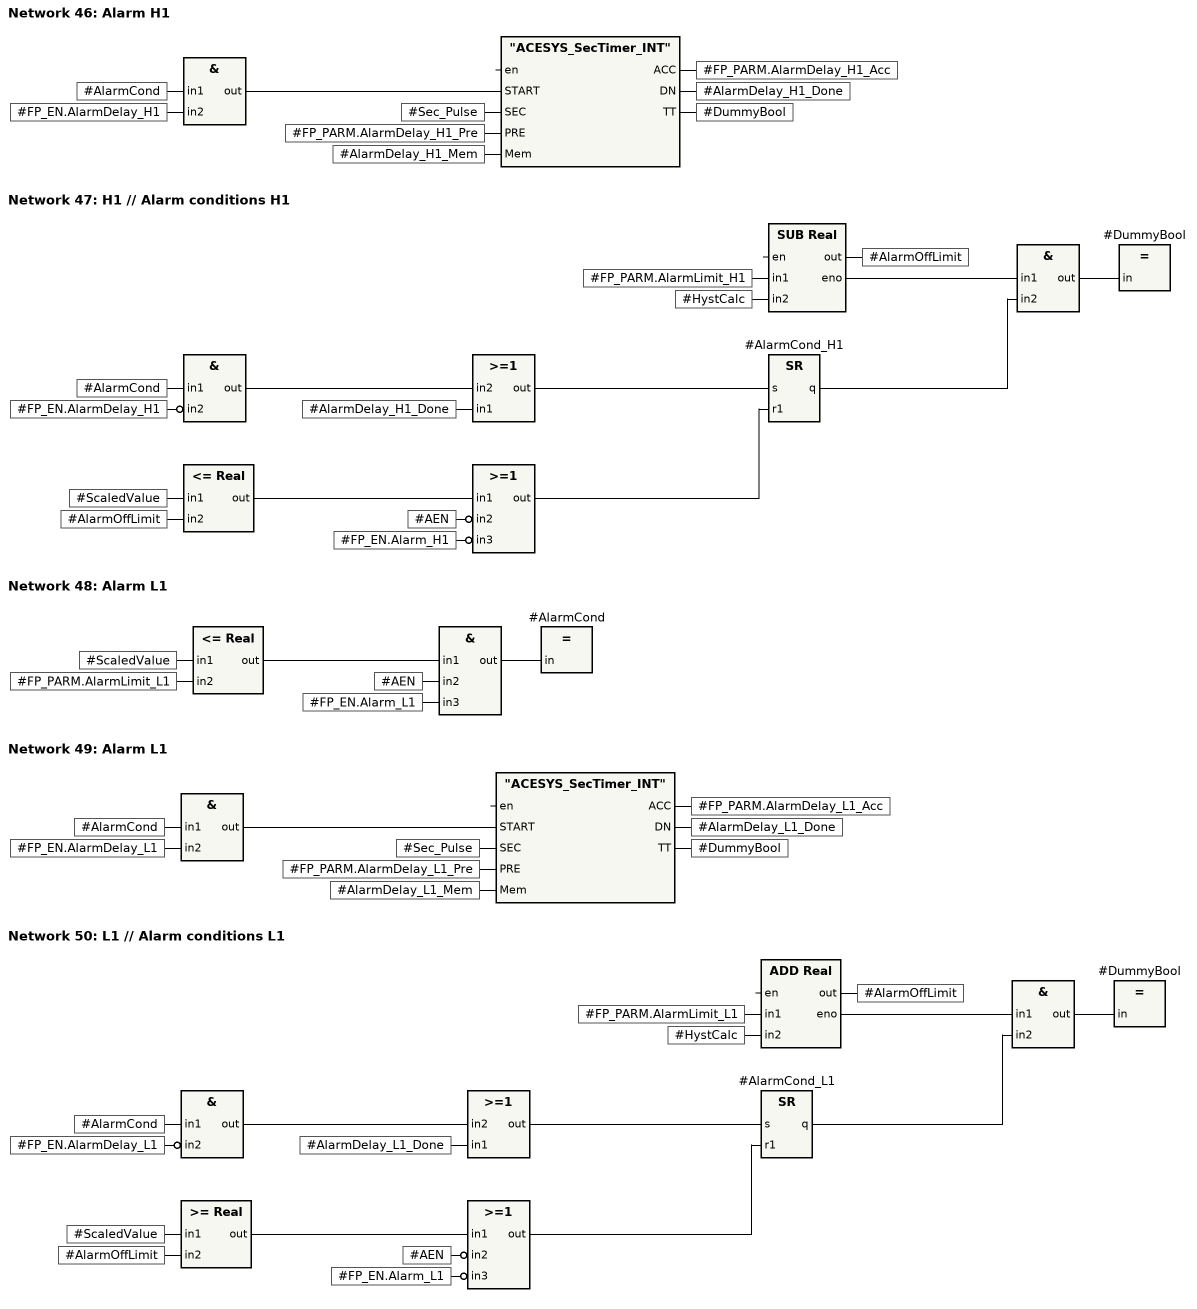
   "ACESYS_SecTimer_INT"(START := #AlarmCond AND #FP_EN.AlarmDelay_H1,
                         SEC := #Sec_Pulse,
                         PRE := #FP_PARM.AlarmDelay_H1_Pre,
                         Mem := #AlarmDelay_H1_Mem,
                         ACC => #FP_PARM.AlarmDelay_H1_Acc,
                         DN => #AlarmDelay_H1_Done,
                         TT => #DummyBool);
END_REGION

REGION Network 47: H1 // Alarm conditions H1
   // ENO of a box is taken as its EN; it also drops when the box reports an error
   #AlarmOffLimit := #FP_PARM.AlarmLimit_H1 - #HystCalc;
   IF (#AlarmCond AND NOT #FP_EN.AlarmDelay_H1) OR #AlarmDelay_H1_Done THEN
       #AlarmCond_H1 := TRUE;   // SR flip-flop
   END_IF;
   IF (#ScaledValue <= #AlarmOffLimit) OR NOT #AEN OR NOT #FP_EN.Alarm_H1 THEN
       #AlarmCond_H1 := FALSE;
   END_IF;
   #DummyBool := #AlarmCond_H1;
END_REGION

REGION Network 48: Alarm L1
   #AlarmCond := (#ScaledValue <= #FP_PARM.AlarmLimit_L1) AND #AEN AND #FP_EN.Alarm_L1;
END_REGION

REGION Network 49: Alarm L1
   "ACESYS_SecTimer_INT"(START := #AlarmCond AND #FP_EN.AlarmDelay_L1,
                         SEC := #Sec_Pulse,
                         PRE := #FP_PARM.AlarmDelay_L1_Pre,
                         Mem := #AlarmDelay_L1_Mem,
                         ACC => #FP_PARM.AlarmDelay_L1_Acc,
                         DN => #AlarmDelay_L1_Done,
                         TT => #DummyBool);
END_REGION

REGION Network 50: L1 // Alarm conditions L1
   // ENO of a box is taken as its EN; it also drops when the box reports an error
   #AlarmOffLimit := #FP_PARM.AlarmLimit_L1 + #HystCalc;
   IF (#AlarmCond AND NOT #FP_EN.AlarmDelay_L1) OR #AlarmDelay_L1_Done THEN
       #AlarmCond_L1 := TRUE;   // SR flip-flop
   END_IF;
   IF (#ScaledValue >= #AlarmOffLimit) OR NOT #AEN OR NOT #FP_EN.Alarm_L1 THEN
       #AlarmCond_L1 := FALSE;
   END_IF;
   #DummyBool := #AlarmCond_L1;
END_REGION

REGION Network 51: Alarm L2
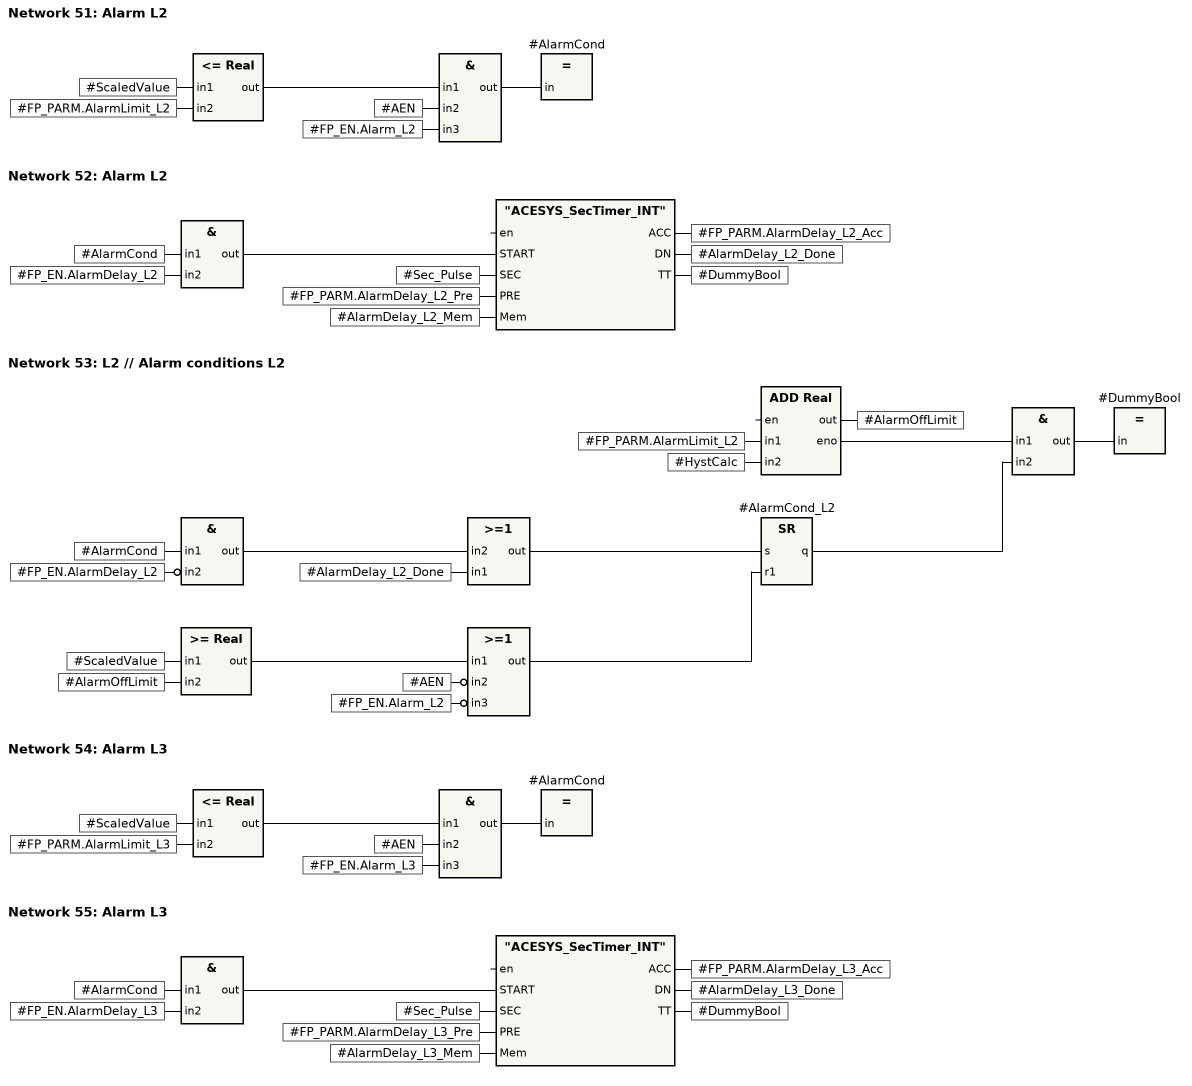
   #AlarmCond := (#ScaledValue <= #FP_PARM.AlarmLimit_L2) AND #AEN AND #FP_EN.Alarm_L2;
END_REGION

REGION Network 52: Alarm L2
   "ACESYS_SecTimer_INT"(START := #AlarmCond AND #FP_EN.AlarmDelay_L2,
                         SEC := #Sec_Pulse,
                         PRE := #FP_PARM.AlarmDelay_L2_Pre,
                         Mem := #AlarmDelay_L2_Mem,
                         ACC => #FP_PARM.AlarmDelay_L2_Acc,
                         DN => #AlarmDelay_L2_Done,
                         TT => #DummyBool);
END_REGION

REGION Network 53: L2 // Alarm conditions L2
   // ENO of a box is taken as its EN; it also drops when the box reports an error
   #AlarmOffLimit := #FP_PARM.AlarmLimit_L2 + #HystCalc;
   IF (#AlarmCond AND NOT #FP_EN.AlarmDelay_L2) OR #AlarmDelay_L2_Done THEN
       #AlarmCond_L2 := TRUE;   // SR flip-flop
   END_IF;
   IF (#ScaledValue >= #AlarmOffLimit) OR NOT #AEN OR NOT #FP_EN.Alarm_L2 THEN
       #AlarmCond_L2 := FALSE;
   END_IF;
   #DummyBool := #AlarmCond_L2;
END_REGION

REGION Network 54: Alarm L3
   #AlarmCond := (#ScaledValue <= #FP_PARM.AlarmLimit_L3) AND #AEN AND #FP_EN.Alarm_L3;
END_REGION

REGION Network 55: Alarm L3
   "ACESYS_SecTimer_INT"(START := #AlarmCond AND #FP_EN.AlarmDelay_L3,
                         SEC := #Sec_Pulse,
                         PRE := #FP_PARM.AlarmDelay_L3_Pre,
                         Mem := #AlarmDelay_L3_Mem,
                         ACC => #FP_PARM.AlarmDelay_L3_Acc,
                         DN => #AlarmDelay_L3_Done,
                         TT => #DummyBool);
END_REGION

REGION Network 56: L3 // Alarm conditions L3
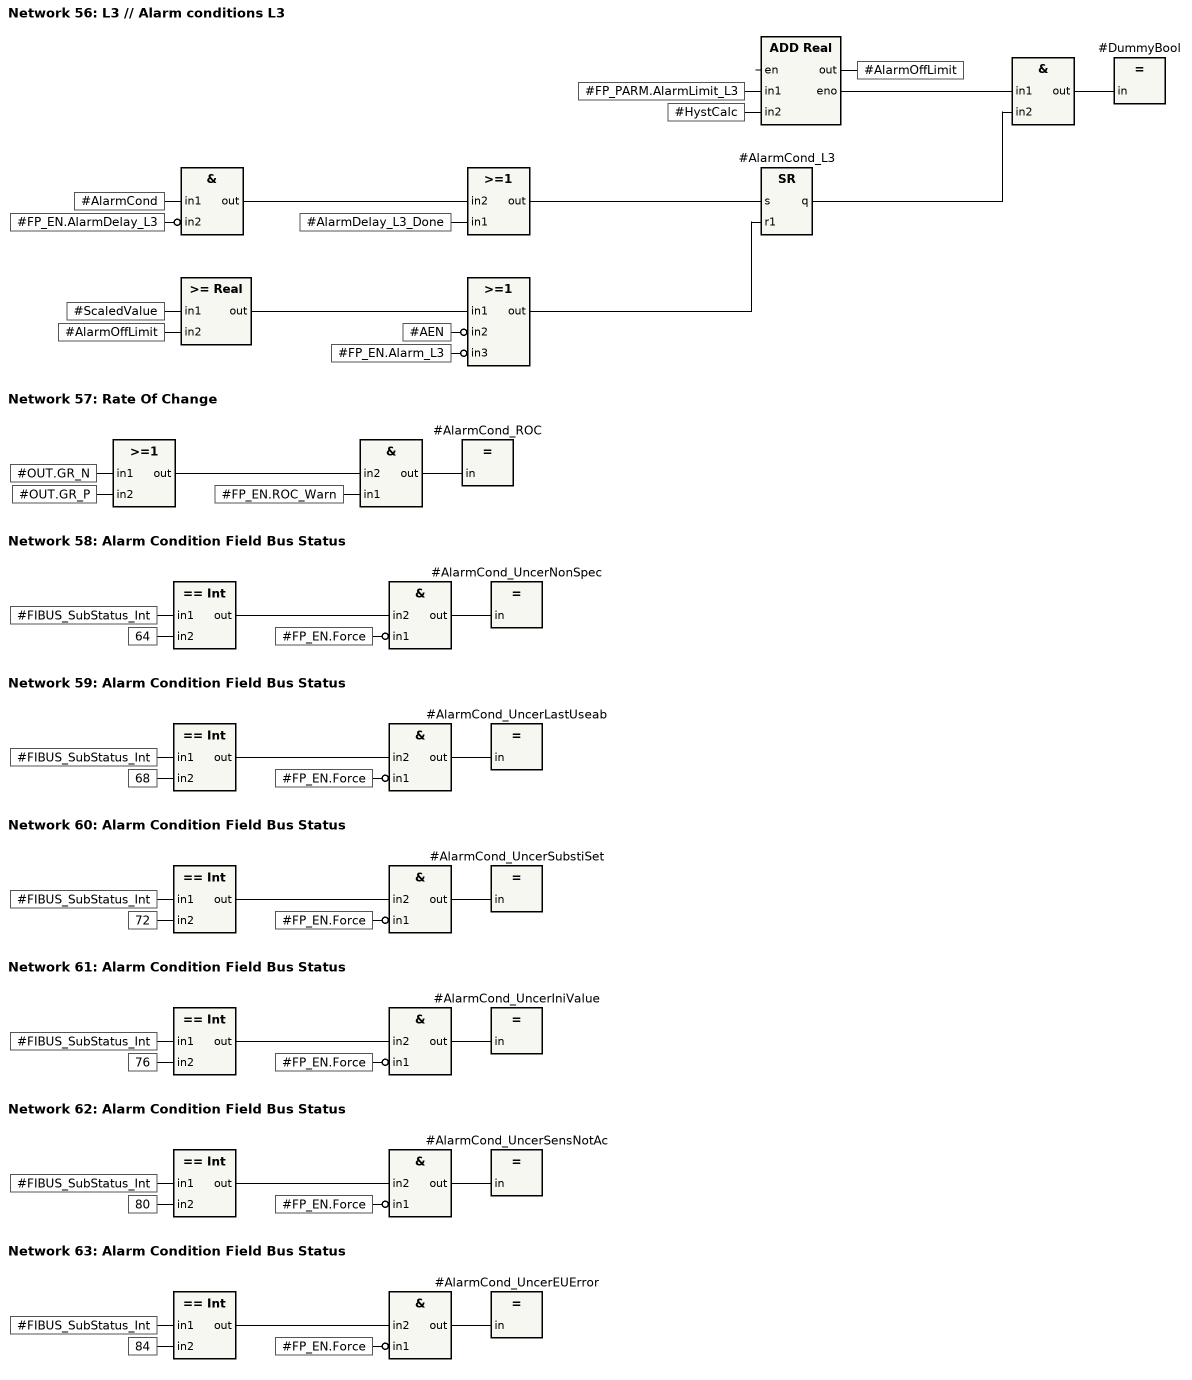
   // ENO of a box is taken as its EN; it also drops when the box reports an error
   #AlarmOffLimit := #FP_PARM.AlarmLimit_L3 + #HystCalc;
   IF (#AlarmCond AND NOT #FP_EN.AlarmDelay_L3) OR #AlarmDelay_L3_Done THEN
       #AlarmCond_L3 := TRUE;   // SR flip-flop
   END_IF;
   IF (#ScaledValue >= #AlarmOffLimit) OR NOT #AEN OR NOT #FP_EN.Alarm_L3 THEN
       #AlarmCond_L3 := FALSE;
   END_IF;
   #DummyBool := #AlarmCond_L3;
END_REGION

REGION Network 57: Rate Of Change
   // >>>>>Rate Of Change (RAC)<<<<<
   // 
   // Warning only
   #AlarmCond_ROC := (#OUT.GR_N OR #OUT.GR_P) AND #FP_EN.ROC_Warn;
END_REGION

REGION Network 58: Alarm Condition Field Bus Status
   // Build 003 - 24 Oct 2019 : FP_En_Force flag added
   #AlarmCond_UncerNonSpec := (#FIBUS_SubStatus_Int = 64) AND NOT #FP_EN.Force;
END_REGION

REGION Network 59: Alarm Condition Field Bus Status
   // Build 003 - 24 Oct 2019 : FP_En_Force flag added
   #AlarmCond_UncerLastUseab := (#FIBUS_SubStatus_Int = 68) AND NOT #FP_EN.Force;
END_REGION

REGION Network 60: Alarm Condition Field Bus Status
   // Build 003 - 24 Oct 2019 : FP_En_Force flag added
   #AlarmCond_UncerSubstiSet := (#FIBUS_SubStatus_Int = 72) AND NOT #FP_EN.Force;
END_REGION

REGION Network 61: Alarm Condition Field Bus Status
   // Build 003 - 24 Oct 2019 : FP_En_Force flag added
   #AlarmCond_UncerIniValue := (#FIBUS_SubStatus_Int = 76) AND NOT #FP_EN.Force;
END_REGION

REGION Network 62: Alarm Condition Field Bus Status
   // Build 003 - 24 Oct 2019 : FP_En_Force flag added
   #AlarmCond_UncerSensNotAc := (#FIBUS_SubStatus_Int = 80) AND NOT #FP_EN.Force;
END_REGION

REGION Network 63: Alarm Condition Field Bus Status
   #AlarmCond_UncerEUError := (#FIBUS_SubStatus_Int = 84) AND NOT #FP_EN.Force;
END_REGION

REGION Network 64: Alarm Condition Field Bus Status
   // Build 003 - 24 Oct 2019 : FP_En_Force flag added
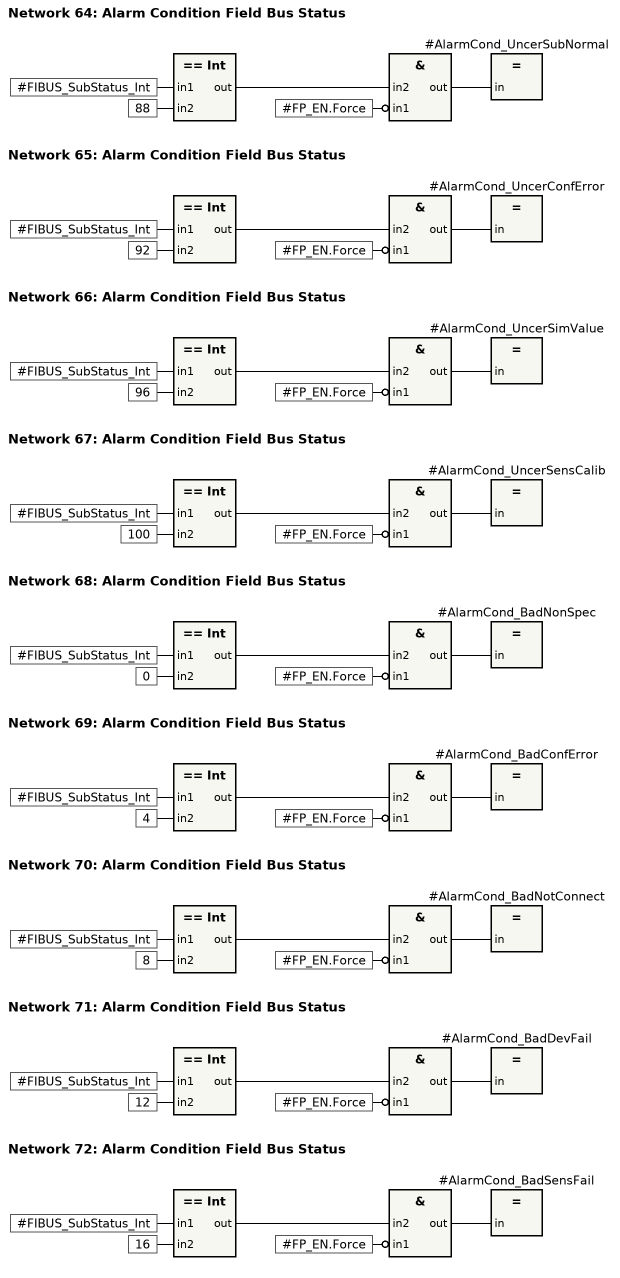
   #AlarmCond_UncerSubNormal := (#FIBUS_SubStatus_Int = 88) AND NOT #FP_EN.Force;
END_REGION

REGION Network 65: Alarm Condition Field Bus Status
   #AlarmCond_UncerConfError := (#FIBUS_SubStatus_Int = 92) AND NOT #FP_EN.Force;
END_REGION

REGION Network 66: Alarm Condition Field Bus Status
   #AlarmCond_UncerSimValue := (#FIBUS_SubStatus_Int = 96) AND NOT #FP_EN.Force;
END_REGION

REGION Network 67: Alarm Condition Field Bus Status
   // Build 003 - 24 Oct 2019 : FP_En_Force flag added
   #AlarmCond_UncerSensCalib := (#FIBUS_SubStatus_Int = 100) AND NOT #FP_EN.Force;
END_REGION

REGION Network 68: Alarm Condition Field Bus Status
   #AlarmCond_BadNonSpec := (#FIBUS_SubStatus_Int = 0) AND NOT #FP_EN.Force;
END_REGION

REGION Network 69: Alarm Condition Field Bus Status
   // Build 003 - 24 Oct 2019 : FP_En_Force flag added
   #AlarmCond_BadConfError := (#FIBUS_SubStatus_Int = 4) AND NOT #FP_EN.Force;
END_REGION

REGION Network 70: Alarm Condition Field Bus Status
   #AlarmCond_BadNotConnect := (#FIBUS_SubStatus_Int = 8) AND NOT #FP_EN.Force;
END_REGION

REGION Network 71: Alarm Condition Field Bus Status
   // Build 003 - 24 Oct 2019 : FP_En_Force flag added
   #AlarmCond_BadDevFail := (#FIBUS_SubStatus_Int = 12) AND NOT #FP_EN.Force;
END_REGION

REGION Network 72: Alarm Condition Field Bus Status
   // Build 003 - 24 Oct 2019 : FP_En_Force flag added
   #AlarmCond_BadSensFail := (#FIBUS_SubStatus_Int = 16) AND NOT #FP_EN.Force;
END_REGION

REGION Network 73: Alarm Condition Field Bus Status
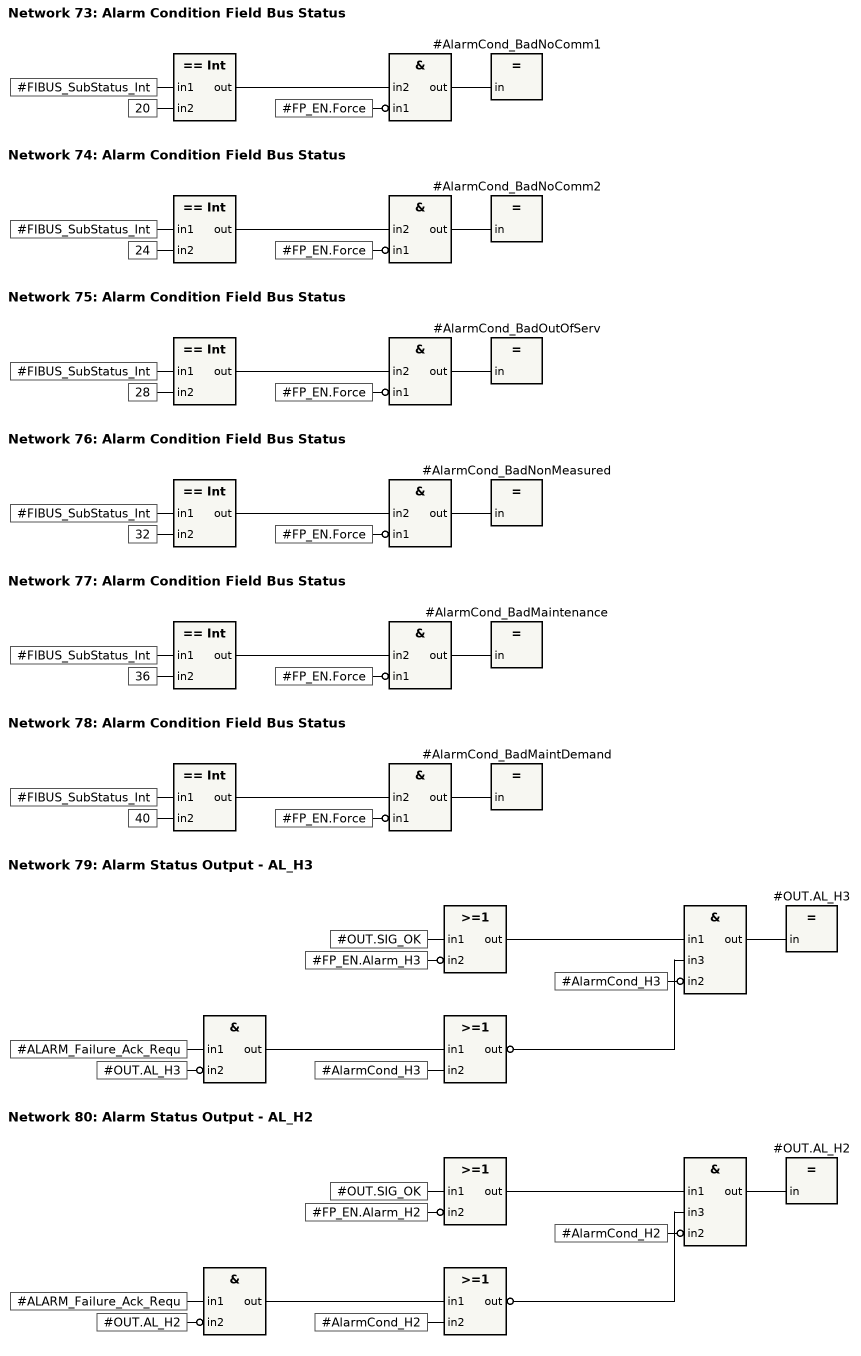
   #AlarmCond_BadNoComm1 := (#FIBUS_SubStatus_Int = 20) AND NOT #FP_EN.Force;
END_REGION

REGION Network 74: Alarm Condition Field Bus Status
   // Build 003 - 24 Oct 2019 : FP_En_Force flag added
   #AlarmCond_BadNoComm2 := (#FIBUS_SubStatus_Int = 24) AND NOT #FP_EN.Force;
END_REGION

REGION Network 75: Alarm Condition Field Bus Status
   #AlarmCond_BadOutOfServ := (#FIBUS_SubStatus_Int = 28) AND NOT #FP_EN.Force;
END_REGION

REGION Network 76: Alarm Condition Field Bus Status
   // Build 003 - 24 Oct 2019 : FP_En_Force flag added
   #AlarmCond_BadNonMeasured := (#FIBUS_SubStatus_Int = 32) AND NOT #FP_EN.Force;
END_REGION

REGION Network 77: Alarm Condition Field Bus Status
   // Build 003 - 24 Oct 2019 : FP_En_Force flag added
   #AlarmCond_BadMaintenance := (#FIBUS_SubStatus_Int = 36) AND NOT #FP_EN.Force;
END_REGION

REGION Network 78: Alarm Condition Field Bus Status
   // Build 003 - 24 Oct 2019 : FP_En_Force flag added
   #AlarmCond_BadMaintDemand := (#FIBUS_SubStatus_Int = 40) AND NOT #FP_EN.Force;
END_REGION

REGION Network 79: Alarm Status Output - AL_H3
   #OUT.AL_H3 := (#OUT.SIG_OK OR NOT #FP_EN.Alarm_H3) AND NOT ((#ALARM_Failure_Ack_Requ AND NOT #OUT.AL_H3) OR #AlarmCond_H3) AND NOT #AlarmCond_H3;
END_REGION

REGION Network 80: Alarm Status Output - AL_H2
   #OUT.AL_H2 := (#OUT.SIG_OK OR NOT #FP_EN.Alarm_H2) AND NOT ((#ALARM_Failure_Ack_Requ AND NOT #OUT.AL_H2) OR #AlarmCond_H2) AND NOT #AlarmCond_H2;
END_REGION

REGION Network 81: Alarm Status Output - AL_H1
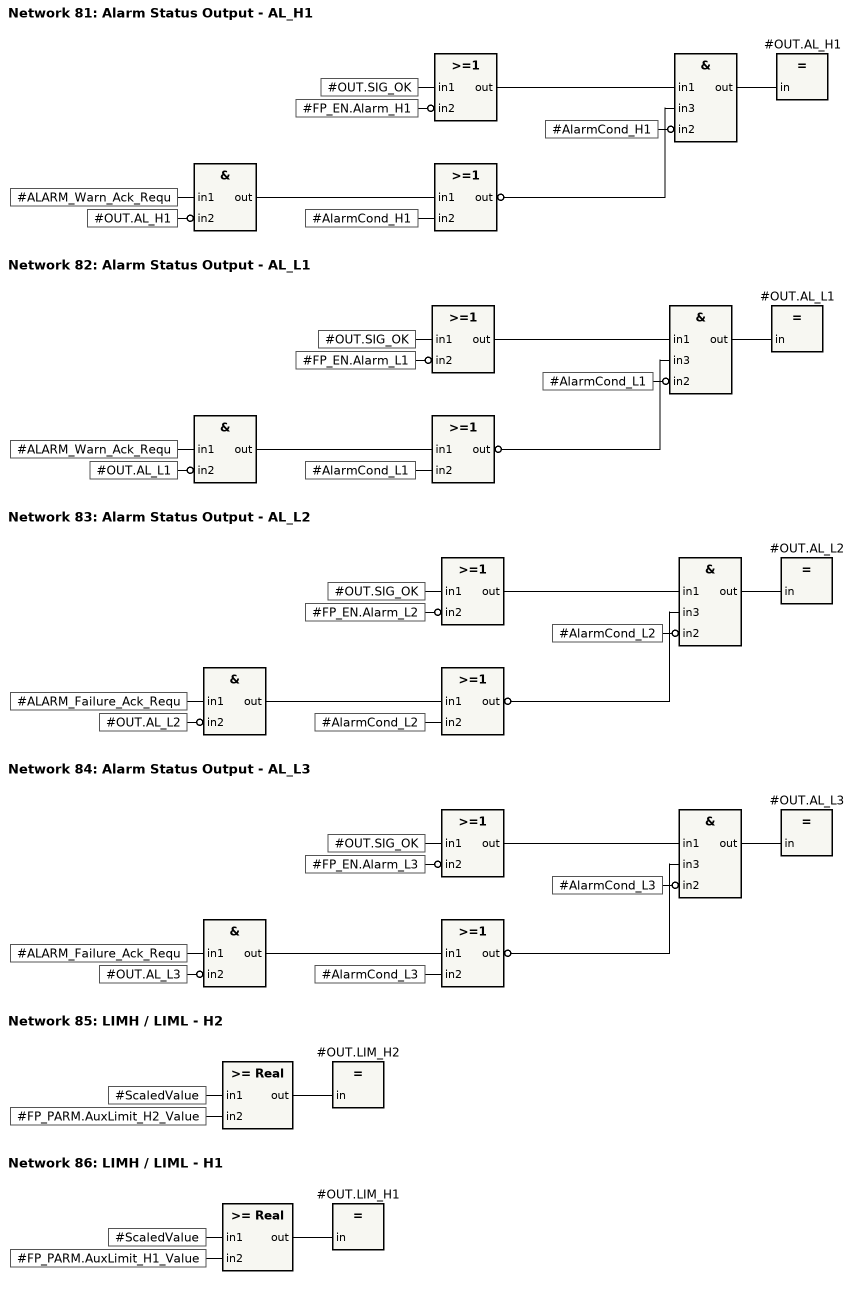
   #OUT.AL_H1 := (#OUT.SIG_OK OR NOT #FP_EN.Alarm_H1) AND NOT ((#ALARM_Warn_Ack_Requ AND NOT #OUT.AL_H1) OR #AlarmCond_H1) AND NOT #AlarmCond_H1;
END_REGION

REGION Network 82: Alarm Status Output - AL_L1
   #OUT.AL_L1 := (#OUT.SIG_OK OR NOT #FP_EN.Alarm_L1) AND NOT ((#ALARM_Warn_Ack_Requ AND NOT #OUT.AL_L1) OR #AlarmCond_L1) AND NOT #AlarmCond_L1;
END_REGION

REGION Network 83: Alarm Status Output - AL_L2
   #OUT.AL_L2 := (#OUT.SIG_OK OR NOT #FP_EN.Alarm_L2) AND NOT ((#ALARM_Failure_Ack_Requ AND NOT #OUT.AL_L2) OR #AlarmCond_L2) AND NOT #AlarmCond_L2;
END_REGION

REGION Network 84: Alarm Status Output - AL_L3
   #OUT.AL_L3 := (#OUT.SIG_OK OR NOT #FP_EN.Alarm_L3) AND NOT ((#ALARM_Failure_Ack_Requ AND NOT #OUT.AL_L3) OR #AlarmCond_L3) AND NOT #AlarmCond_L3;
END_REGION

REGION Network 85: LIMH / LIML - H2
   #OUT.LIM_H2 := #ScaledValue >= #FP_PARM.AuxLimit_H2_Value;
END_REGION

REGION Network 86: LIMH / LIML - H1
   #OUT.LIM_H1 := #ScaledValue >= #FP_PARM.AuxLimit_H1_Value;
END_REGION

REGION Network 87: LIMH / LIML - L1
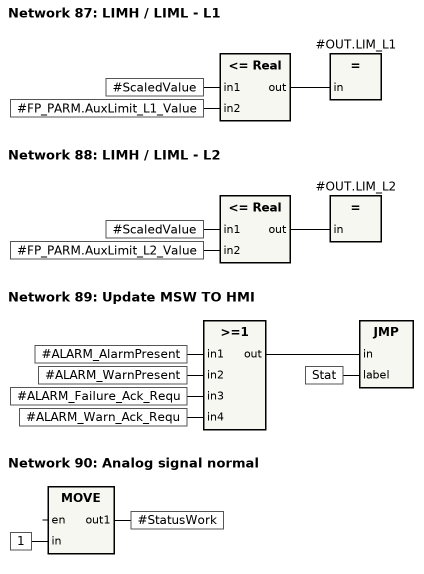
   #OUT.LIM_L1 := #ScaledValue <= #FP_PARM.AuxLimit_L1_Value;
END_REGION

REGION Network 88: LIMH / LIML - L2
   #OUT.LIM_L2 := #ScaledValue <= #FP_PARM.AuxLimit_L2_Value;
END_REGION

REGION Network 89: Update MSW TO HMI
   // Stat = Skip Sensor Status
   IF #ALARM_AlarmPresent OR #ALARM_WarnPresent OR #ALARM_Failure_Ack_Requ OR #ALARM_Warn_Ack_Requ THEN
       GOTO Stat;
   END_IF;
END_REGION

REGION Network 90: Analog signal normal
   #StatusWork := 1;
END_REGION

REGION Network 91: Report Good status
   // 132 = Active block alarm
   // 136 = Active advisory alarm
   // 140 = Active critical alarm
   // 144 = Unacknowledged block alarm
   // 148 = Unacknowledged advisory alarm
   // 152 = Unacknowledged critical alarm
   // 156 = Not used
   // 160 = Init fail safe
   // 164 = Maintenance required
   // 
   // Build 006 - 22 Nov 2017 : Status work changed from 132 - 164 to 50 - 57
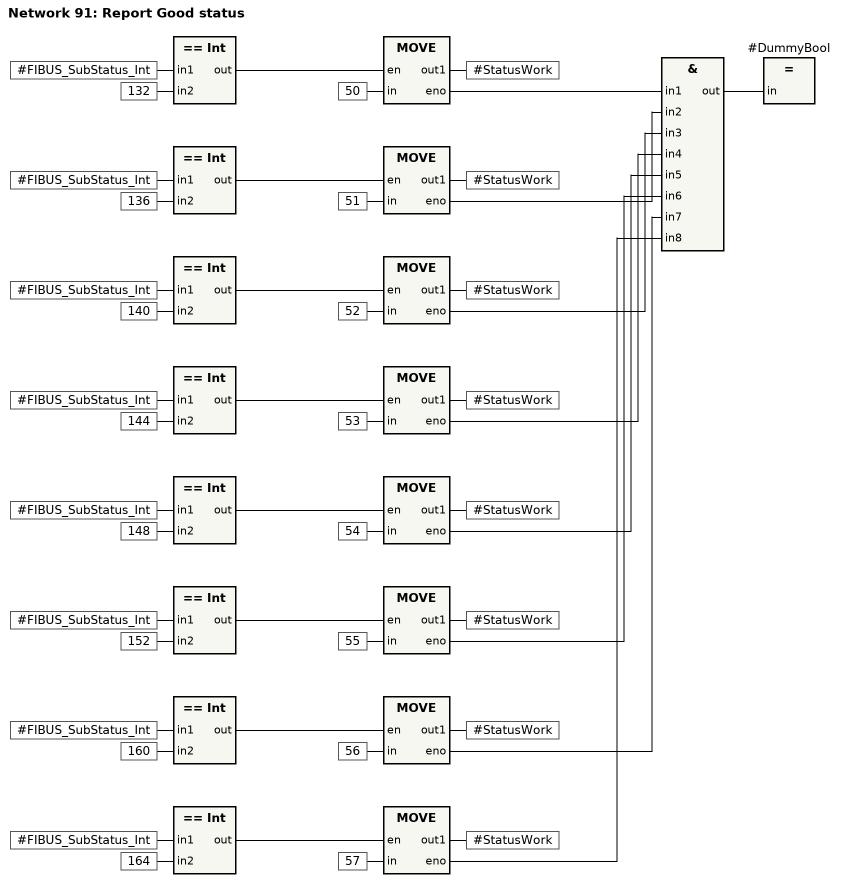
   // ENO of a box is taken as its EN; it also drops when the box reports an error
   #_w1 := #FIBUS_SubStatus_Int = 132;
   IF #_w1 THEN #StatusWork := 50; END_IF;
   #_w2 := #FIBUS_SubStatus_Int = 136;
   IF #_w2 THEN #StatusWork := 51; END_IF;
   #_w3 := #FIBUS_SubStatus_Int = 140;
   IF #_w3 THEN #StatusWork := 52; END_IF;
   #_w4 := #FIBUS_SubStatus_Int = 144;
   IF #_w4 THEN #StatusWork := 53; END_IF;
   #_w5 := #FIBUS_SubStatus_Int = 148;
   IF #_w5 THEN #StatusWork := 54; END_IF;
   #_w6 := #FIBUS_SubStatus_Int = 152;
   IF #_w6 THEN #StatusWork := 55; END_IF;
   #_w7 := #FIBUS_SubStatus_Int = 160;
   IF #_w7 THEN #StatusWork := 56; END_IF;
   #_w8 := #FIBUS_SubStatus_Int = 164;
   IF #_w8 THEN #StatusWork := 57; END_IF;
   #DummyBool := #_w1 AND #_w2 AND #_w3 AND #_w4 AND #_w5 AND #_w6 AND #_w7 AND #_w8;
END_REGION

REGION Network 92: Jump Network
   // >>>>>SIGNAL VALID DETECTION<<<<<
   // 
   // Jump destination if ignore sensor Status
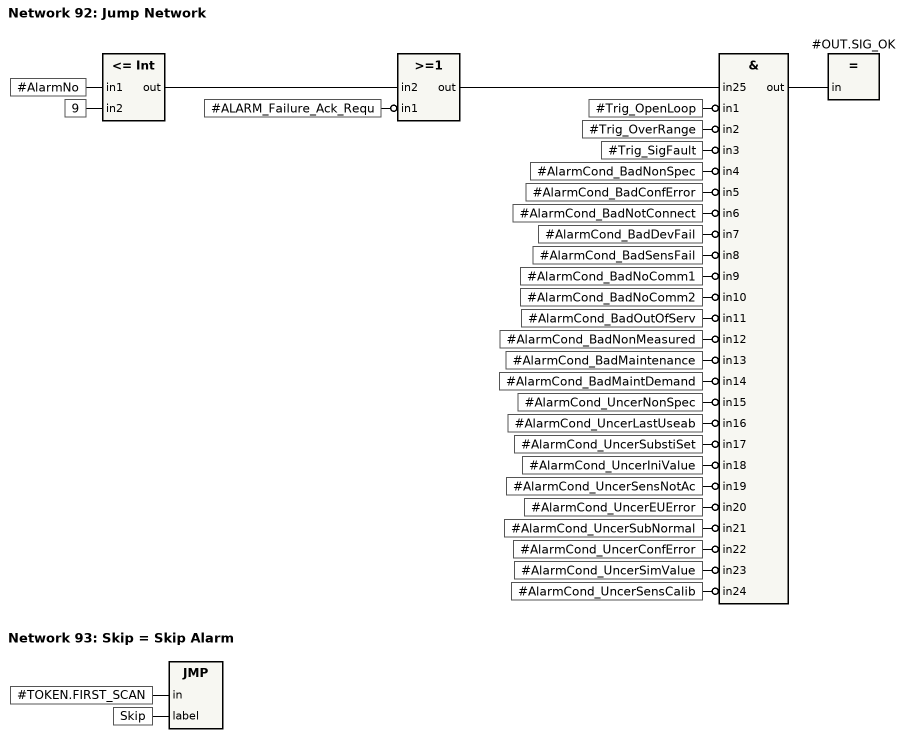
   Stat:
   #OUT.SIG_OK := ((#AlarmNo <= 9) OR NOT #ALARM_Failure_Ack_Requ) AND NOT #Trig_OpenLoop AND NOT #Trig_OverRange AND NOT #Trig_SigFault AND NOT #AlarmCond_BadNonSpec AND NOT #AlarmCond_BadConfError AND NOT #AlarmCond_BadNotConnect AND NOT #AlarmCond_BadDevFail AND NOT #AlarmCond_BadSensFail AND NOT #AlarmCond_BadNoComm1 AND NOT #AlarmCond_BadNoComm2 AND NOT #AlarmCond_BadOutOfServ AND NOT #AlarmCond_BadNonMeasured AND NOT #AlarmCond_BadMaintenance AND NOT #AlarmCond_BadMaintDemand AND NOT #AlarmCond_UncerNonSpec AND NOT #AlarmCond_UncerLastUseab AND NOT #AlarmCond_UncerSubstiSet AND NOT #AlarmCond_UncerIniValue AND NOT #AlarmCond_UncerSensNotAc AND NOT #AlarmCond_UncerEUError AND NOT #AlarmCond_UncerSubNormal AND NOT #AlarmCond_UncerConfError AND NOT #AlarmCond_UncerSimValue AND NOT #AlarmCond_UncerSensCalib;
END_REGION

REGION Network 93: Skip = Skip Alarm
   // >>>>>Alarm Present<<<<<
   // 
   // Skip = Skip Alarm
   IF #TOKEN.FIRST_SCAN THEN GOTO Skip; END_IF;
END_REGION

REGION Network 94: Alarm
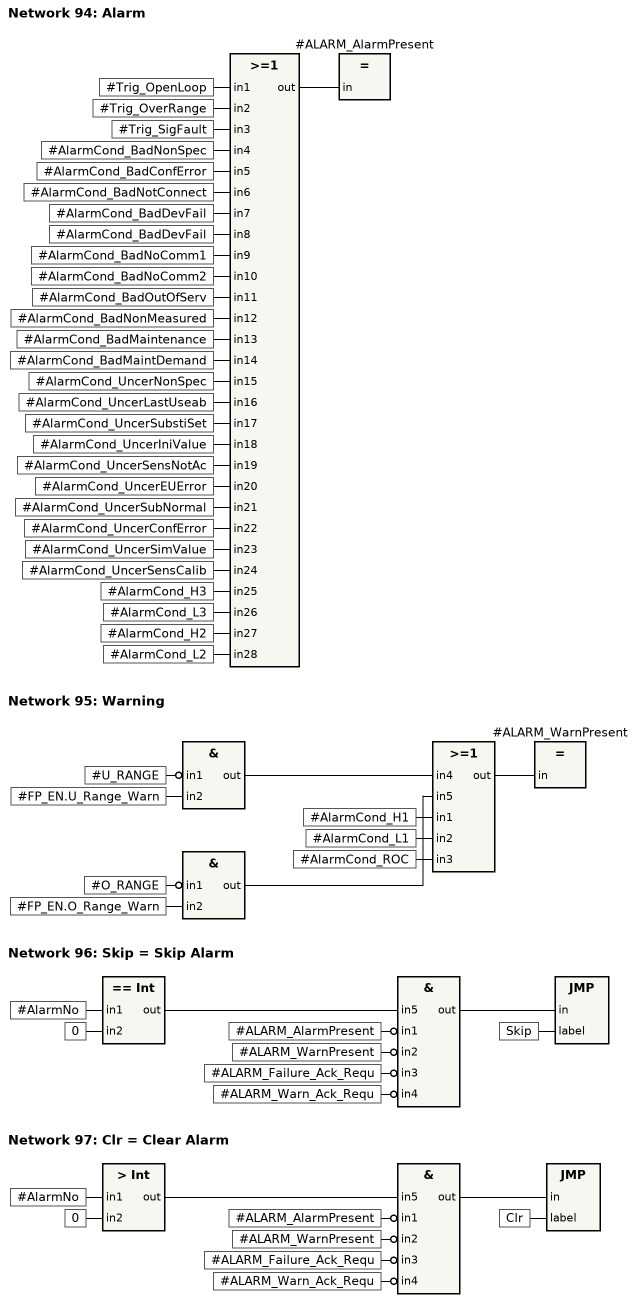
   #ALARM_AlarmPresent := #Trig_OpenLoop OR #Trig_OverRange OR #Trig_SigFault OR #AlarmCond_BadNonSpec OR #AlarmCond_BadConfError OR #AlarmCond_BadNotConnect OR #AlarmCond_BadDevFail OR #AlarmCond_BadDevFail OR #AlarmCond_BadNoComm1 OR #AlarmCond_BadNoComm2 OR #AlarmCond_BadOutOfServ OR #AlarmCond_BadNonMeasured OR #AlarmCond_BadMaintenance OR #AlarmCond_BadMaintDemand OR #AlarmCond_UncerNonSpec OR #AlarmCond_UncerLastUseab OR #AlarmCond_UncerSubstiSet OR #AlarmCond_UncerIniValue OR #AlarmCond_UncerSensNotAc OR #AlarmCond_UncerEUError OR #AlarmCond_UncerSubNormal OR #AlarmCond_UncerConfError OR #AlarmCond_UncerSimValue OR #AlarmCond_UncerSensCalib OR #AlarmCond_H3 OR #AlarmCond_L3 OR #AlarmCond_H2 OR #AlarmCond_L2;
END_REGION

REGION Network 95: Warning
   #ALARM_WarnPresent := (NOT #U_RANGE AND #FP_EN.U_Range_Warn) OR (NOT #O_RANGE AND #FP_EN.O_Range_Warn) OR #AlarmCond_H1 OR #AlarmCond_L1 OR #AlarmCond_ROC;
END_REGION

REGION Network 96: Skip = Skip Alarm
   IF (#AlarmNo = 0) AND NOT #ALARM_AlarmPresent AND NOT #ALARM_WarnPresent AND NOT #ALARM_Failure_Ack_Requ AND NOT #ALARM_Warn_Ack_Requ THEN
       GOTO Skip;
   END_IF;
END_REGION

REGION Network 97: Clr = Clear Alarm
   IF (#AlarmNo > 0) AND NOT #ALARM_AlarmPresent AND NOT #ALARM_WarnPresent AND NOT #ALARM_Failure_Ack_Requ AND NOT #ALARM_Warn_Ack_Requ THEN
       GOTO Clr;
   END_IF;
END_REGION

REGION Network 98: Ack = Alarm Acknowledge
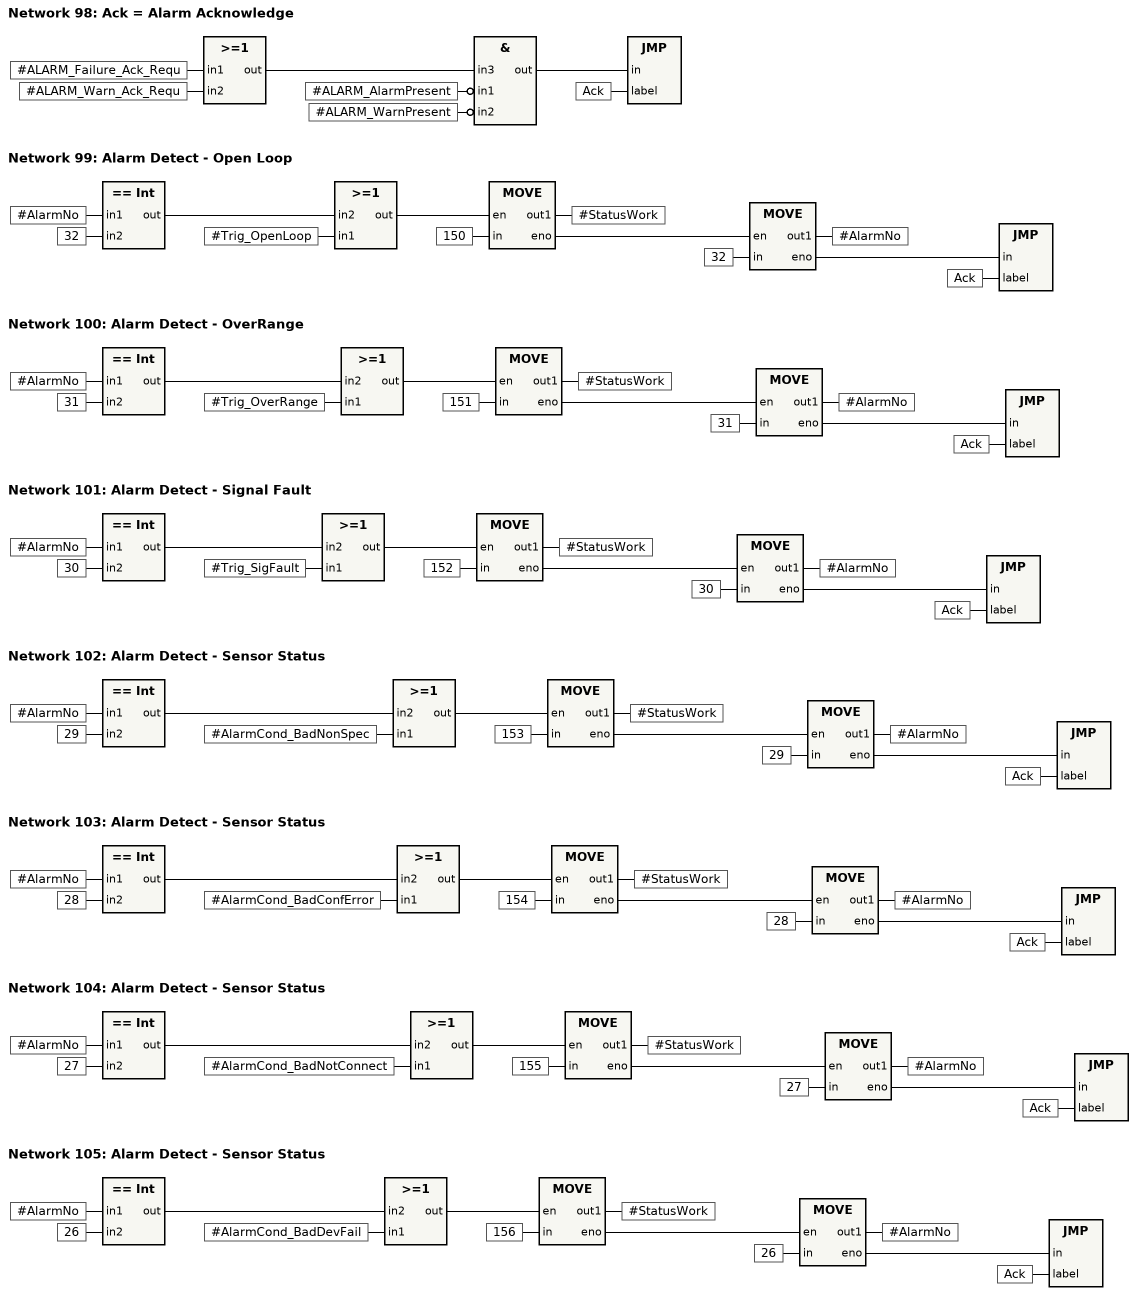
   IF (#ALARM_Failure_Ack_Requ OR #ALARM_Warn_Ack_Requ) AND NOT #ALARM_AlarmPresent AND NOT #ALARM_WarnPresent THEN
       GOTO Ack;
   END_IF;
END_REGION

REGION Network 99: Alarm Detect - Open Loop
   // ENO of a box is taken as its EN; it also drops when the box reports an error
   #_w1 := (#AlarmNo = 32) OR #Trig_OpenLoop;
   IF #_w1 THEN
       #StatusWork := 150;
       #AlarmNo := 32;
       GOTO Ack;
   END_IF;
END_REGION

REGION Network 100: Alarm Detect - OverRange
   // ENO of a box is taken as its EN; it also drops when the box reports an error
   #_w1 := (#AlarmNo = 31) OR #Trig_OverRange;
   IF #_w1 THEN
       #StatusWork := 151;
       #AlarmNo := 31;
       GOTO Ack;
   END_IF;
END_REGION

REGION Network 101: Alarm Detect - Signal Fault
   // ENO of a box is taken as its EN; it also drops when the box reports an error
   #_w1 := (#AlarmNo = 30) OR #Trig_SigFault;
   IF #_w1 THEN
       #StatusWork := 152;
       #AlarmNo := 30;
       GOTO Ack;
   END_IF;
END_REGION

REGION Network 102: Alarm Detect - Sensor Status
   // ENO of a box is taken as its EN; it also drops when the box reports an error
   #_w1 := (#AlarmNo = 29) OR #AlarmCond_BadNonSpec;
   IF #_w1 THEN
       #StatusWork := 153;
       #AlarmNo := 29;
       GOTO Ack;
   END_IF;
END_REGION

REGION Network 103: Alarm Detect - Sensor Status
   // ENO of a box is taken as its EN; it also drops when the box reports an error
   #_w1 := (#AlarmNo = 28) OR #AlarmCond_BadConfError;
   IF #_w1 THEN
       #StatusWork := 154;
       #AlarmNo := 28;
       GOTO Ack;
   END_IF;
END_REGION

REGION Network 104: Alarm Detect - Sensor Status
   // ENO of a box is taken as its EN; it also drops when the box reports an error
   #_w1 := (#AlarmNo = 27) OR #AlarmCond_BadNotConnect;
   IF #_w1 THEN
       #StatusWork := 155;
       #AlarmNo := 27;
       GOTO Ack;
   END_IF;
END_REGION

REGION Network 105: Alarm Detect - Sensor Status
   // ENO of a box is taken as its EN; it also drops when the box reports an error
   #_w1 := (#AlarmNo = 26) OR #AlarmCond_BadDevFail;
   IF #_w1 THEN
       #StatusWork := 156;
       #AlarmNo := 26;
       GOTO Ack;
   END_IF;
END_REGION

REGION Network 106: Alarm Detect - Sensor Status
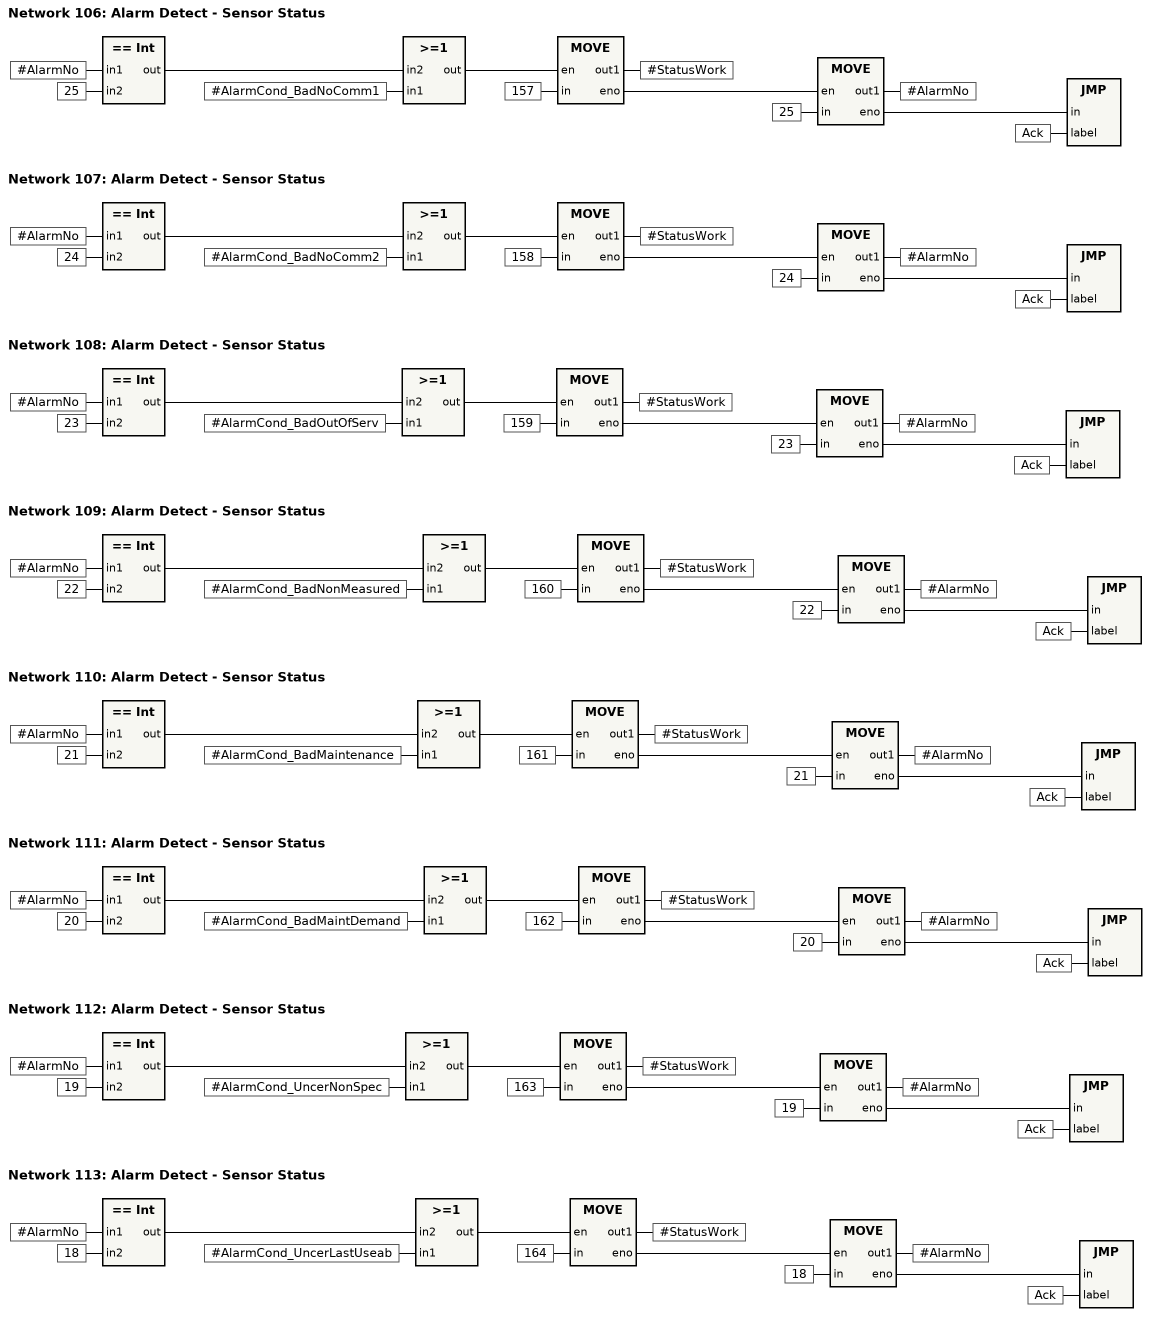
   // ENO of a box is taken as its EN; it also drops when the box reports an error
   #_w1 := (#AlarmNo = 25) OR #AlarmCond_BadNoComm1;
   IF #_w1 THEN
       #StatusWork := 157;
       #AlarmNo := 25;
       GOTO Ack;
   END_IF;
END_REGION

REGION Network 107: Alarm Detect - Sensor Status
   // ENO of a box is taken as its EN; it also drops when the box reports an error
   #_w1 := (#AlarmNo = 24) OR #AlarmCond_BadNoComm2;
   IF #_w1 THEN
       #StatusWork := 158;
       #AlarmNo := 24;
       GOTO Ack;
   END_IF;
END_REGION

REGION Network 108: Alarm Detect - Sensor Status
   // ENO of a box is taken as its EN; it also drops when the box reports an error
   #_w1 := (#AlarmNo = 23) OR #AlarmCond_BadOutOfServ;
   IF #_w1 THEN
       #StatusWork := 159;
       #AlarmNo := 23;
       GOTO Ack;
   END_IF;
END_REGION

REGION Network 109: Alarm Detect - Sensor Status
   // ENO of a box is taken as its EN; it also drops when the box reports an error
   #_w1 := (#AlarmNo = 22) OR #AlarmCond_BadNonMeasured;
   IF #_w1 THEN
       #StatusWork := 160;
       #AlarmNo := 22;
       GOTO Ack;
   END_IF;
END_REGION

REGION Network 110: Alarm Detect - Sensor Status
   // ENO of a box is taken as its EN; it also drops when the box reports an error
   #_w1 := (#AlarmNo = 21) OR #AlarmCond_BadMaintenance;
   IF #_w1 THEN
       #StatusWork := 161;
       #AlarmNo := 21;
       GOTO Ack;
   END_IF;
END_REGION

REGION Network 111: Alarm Detect - Sensor Status
   // ENO of a box is taken as its EN; it also drops when the box reports an error
   #_w1 := (#AlarmNo = 20) OR #AlarmCond_BadMaintDemand;
   IF #_w1 THEN
       #StatusWork := 162;
       #AlarmNo := 20;
       GOTO Ack;
   END_IF;
END_REGION

REGION Network 112: Alarm Detect - Sensor Status
   // ENO of a box is taken as its EN; it also drops when the box reports an error
   #_w1 := (#AlarmNo = 19) OR #AlarmCond_UncerNonSpec;
   IF #_w1 THEN
       #StatusWork := 163;
       #AlarmNo := 19;
       GOTO Ack;
   END_IF;
END_REGION

REGION Network 113: Alarm Detect - Sensor Status
   // ENO of a box is taken as its EN; it also drops when the box reports an error
   #_w1 := (#AlarmNo = 18) OR #AlarmCond_UncerLastUseab;
   IF #_w1 THEN
       #StatusWork := 164;
       #AlarmNo := 18;
       GOTO Ack;
   END_IF;
END_REGION

REGION Network 114: Alarm Detect - Sensor Status
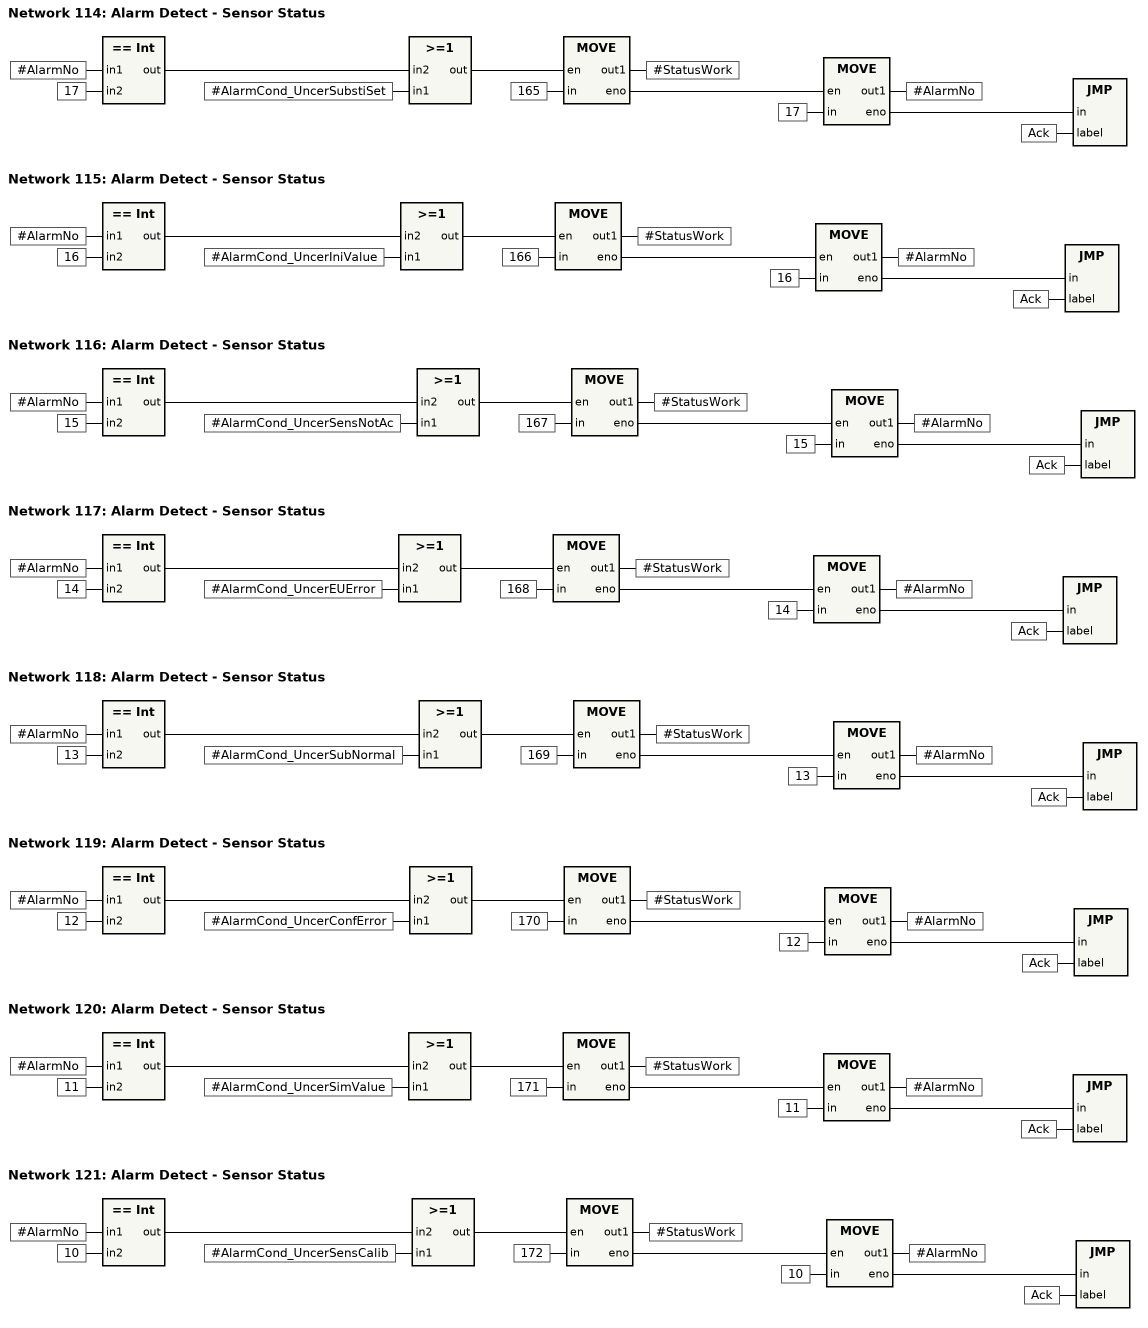
   // ENO of a box is taken as its EN; it also drops when the box reports an error
   #_w1 := (#AlarmNo = 17) OR #AlarmCond_UncerSubstiSet;
   IF #_w1 THEN
       #StatusWork := 165;
       #AlarmNo := 17;
       GOTO Ack;
   END_IF;
END_REGION

REGION Network 115: Alarm Detect - Sensor Status
   // ENO of a box is taken as its EN; it also drops when the box reports an error
   #_w1 := (#AlarmNo = 16) OR #AlarmCond_UncerIniValue;
   IF #_w1 THEN
       #StatusWork := 166;
       #AlarmNo := 16;
       GOTO Ack;
   END_IF;
END_REGION

REGION Network 116: Alarm Detect - Sensor Status
   // ENO of a box is taken as its EN; it also drops when the box reports an error
   #_w1 := (#AlarmNo = 15) OR #AlarmCond_UncerSensNotAc;
   IF #_w1 THEN
       #StatusWork := 167;
       #AlarmNo := 15;
       GOTO Ack;
   END_IF;
END_REGION

REGION Network 117: Alarm Detect - Sensor Status
   // ENO of a box is taken as its EN; it also drops when the box reports an error
   #_w1 := (#AlarmNo = 14) OR #AlarmCond_UncerEUError;
   IF #_w1 THEN
       #StatusWork := 168;
       #AlarmNo := 14;
       GOTO Ack;
   END_IF;
END_REGION

REGION Network 118: Alarm Detect - Sensor Status
   // ENO of a box is taken as its EN; it also drops when the box reports an error
   #_w1 := (#AlarmNo = 13) OR #AlarmCond_UncerSubNormal;
   IF #_w1 THEN
       #StatusWork := 169;
       #AlarmNo := 13;
       GOTO Ack;
   END_IF;
END_REGION

REGION Network 119: Alarm Detect - Sensor Status
   // ENO of a box is taken as its EN; it also drops when the box reports an error
   #_w1 := (#AlarmNo = 12) OR #AlarmCond_UncerConfError;
   IF #_w1 THEN
       #StatusWork := 170;
       #AlarmNo := 12;
       GOTO Ack;
   END_IF;
END_REGION

REGION Network 120: Alarm Detect - Sensor Status
   // ENO of a box is taken as its EN; it also drops when the box reports an error
   #_w1 := (#AlarmNo = 11) OR #AlarmCond_UncerSimValue;
   IF #_w1 THEN
       #StatusWork := 171;
       #AlarmNo := 11;
       GOTO Ack;
   END_IF;
END_REGION

REGION Network 121: Alarm Detect - Sensor Status
   // ENO of a box is taken as its EN; it also drops when the box reports an error
   #_w1 := (#AlarmNo = 10) OR #AlarmCond_UncerSensCalib;
   IF #_w1 THEN
       #StatusWork := 172;
       #AlarmNo := 10;
       GOTO Ack;
   END_IF;
END_REGION

REGION Network 122: Alarm Detect - Alarm H3
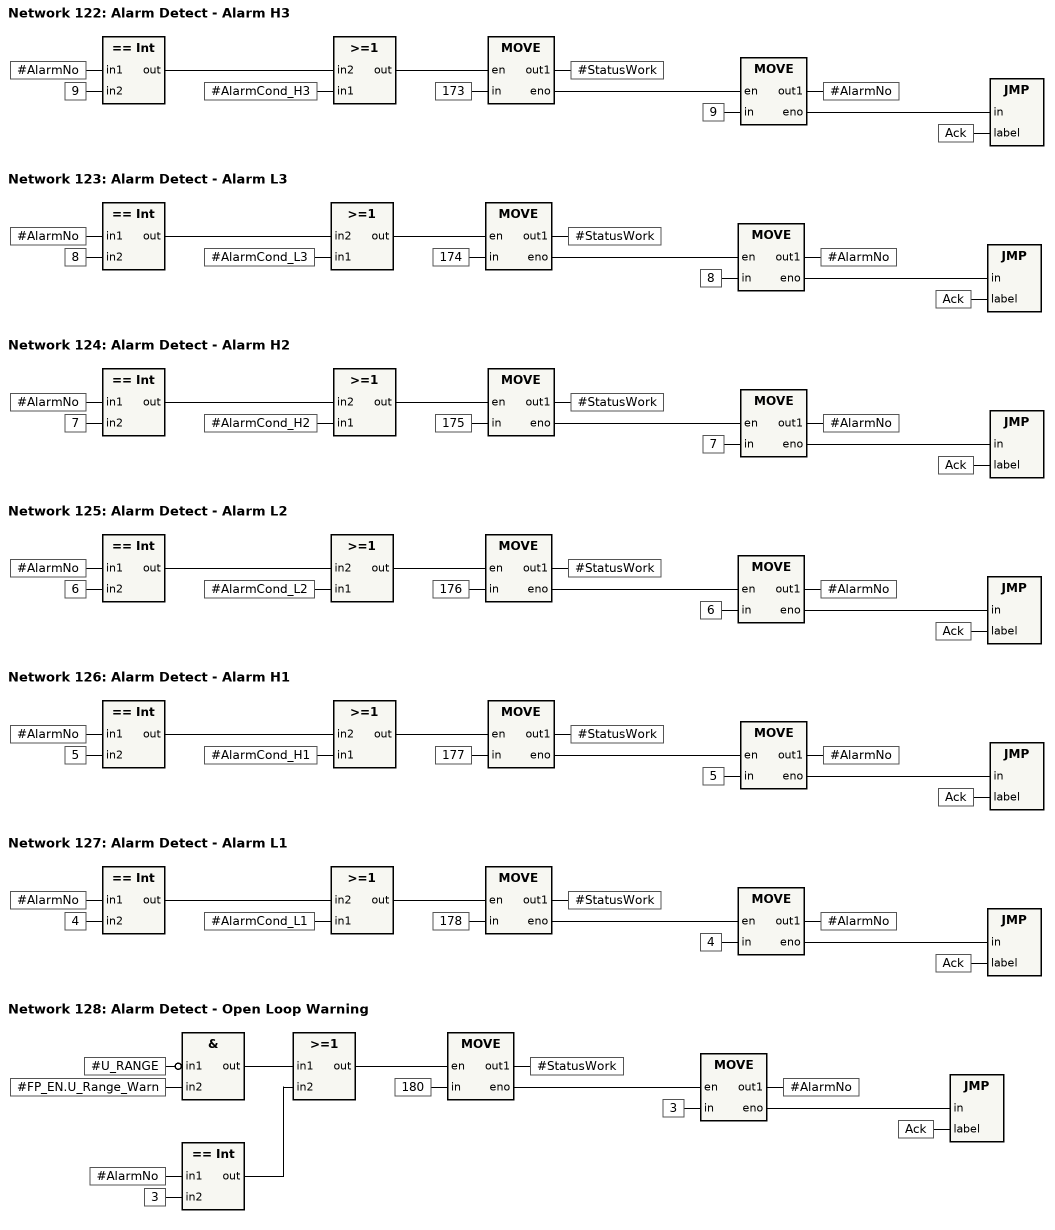
   // ENO of a box is taken as its EN; it also drops when the box reports an error
   #_w1 := (#AlarmNo = 9) OR #AlarmCond_H3;
   IF #_w1 THEN
       #StatusWork := 173;
       #AlarmNo := 9;
       GOTO Ack;
   END_IF;
END_REGION

REGION Network 123: Alarm Detect - Alarm L3
   // ENO of a box is taken as its EN; it also drops when the box reports an error
   #_w1 := (#AlarmNo = 8) OR #AlarmCond_L3;
   IF #_w1 THEN
       #StatusWork := 174;
       #AlarmNo := 8;
       GOTO Ack;
   END_IF;
END_REGION

REGION Network 124: Alarm Detect - Alarm H2
   // ENO of a box is taken as its EN; it also drops when the box reports an error
   #_w1 := (#AlarmNo = 7) OR #AlarmCond_H2;
   IF #_w1 THEN
       #StatusWork := 175;
       #AlarmNo := 7;
       GOTO Ack;
   END_IF;
END_REGION

REGION Network 125: Alarm Detect - Alarm L2
   // ENO of a box is taken as its EN; it also drops when the box reports an error
   #_w1 := (#AlarmNo = 6) OR #AlarmCond_L2;
   IF #_w1 THEN
       #StatusWork := 176;
       #AlarmNo := 6;
       GOTO Ack;
   END_IF;
END_REGION

REGION Network 126: Alarm Detect - Alarm H1
   // ENO of a box is taken as its EN; it also drops when the box reports an error
   #_w1 := (#AlarmNo = 5) OR #AlarmCond_H1;
   IF #_w1 THEN
       #StatusWork := 177;
       #AlarmNo := 5;
       GOTO Ack;
   END_IF;
END_REGION

REGION Network 127: Alarm Detect - Alarm L1
   // ENO of a box is taken as its EN; it also drops when the box reports an error
   #_w1 := (#AlarmNo = 4) OR #AlarmCond_L1;
   IF #_w1 THEN
       #StatusWork := 178;
       #AlarmNo := 4;
       GOTO Ack;
   END_IF;
END_REGION

REGION Network 128: Alarm Detect - Open Loop Warning
   // ENO of a box is taken as its EN; it also drops when the box reports an error
   #_w1 := (NOT #U_RANGE AND #FP_EN.U_Range_Warn) OR (#AlarmNo = 3);
   IF #_w1 THEN
       #StatusWork := 180;
       #AlarmNo := 3;
       GOTO Ack;
   END_IF;
END_REGION

REGION Network 129: Alarm Detect - Short Circiut Warning
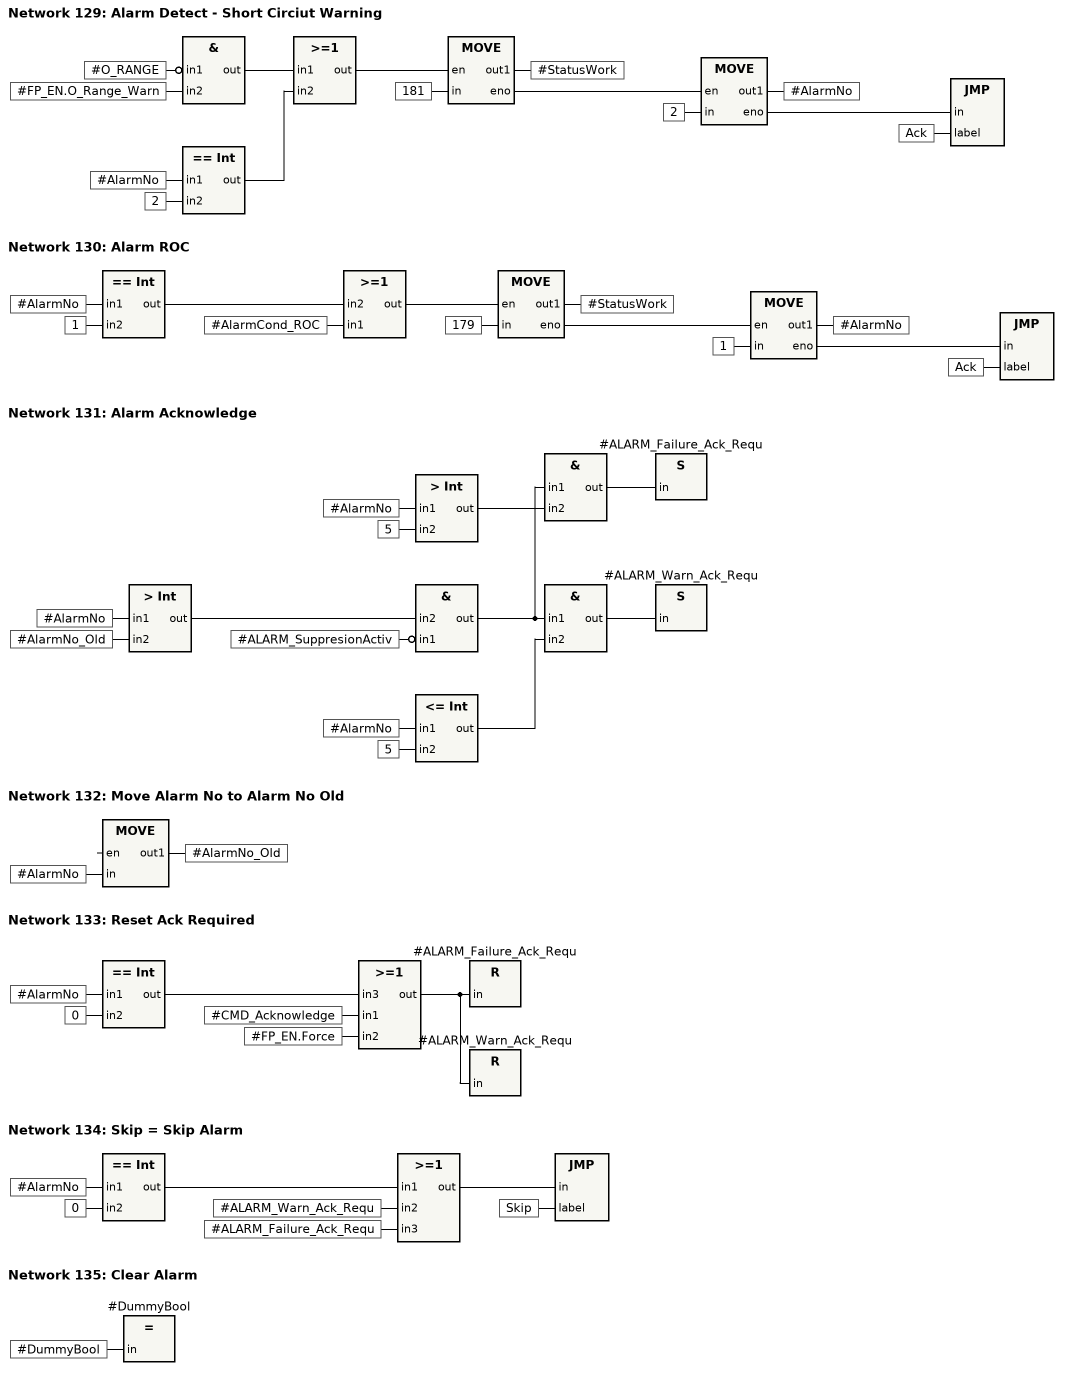
   // ENO of a box is taken as its EN; it also drops when the box reports an error
   #_w1 := (NOT #O_RANGE AND #FP_EN.O_Range_Warn) OR (#AlarmNo = 2);
   IF #_w1 THEN
       #StatusWork := 181;
       #AlarmNo := 2;
       GOTO Ack;
   END_IF;
END_REGION

REGION Network 130: Alarm ROC
   // ENO of a box is taken as its EN; it also drops when the box reports an error
   #_w1 := (#AlarmNo = 1) OR #AlarmCond_ROC;
   IF #_w1 THEN
       #StatusWork := 179;
       #AlarmNo := 1;
       GOTO Ack;
   END_IF;
END_REGION

REGION Network 131: Alarm Acknowledge
   Ack:
   #_w1 := (#AlarmNo > #AlarmNo_Old) AND NOT #ALARM_SuppresionActiv;
   IF #_w1 AND (#AlarmNo > 5) THEN #ALARM_Failure_Ack_Requ := TRUE; END_IF;
   IF #_w1 AND (#AlarmNo <= 5) THEN #ALARM_Warn_Ack_Requ := TRUE; END_IF;
END_REGION

REGION Network 132: Move Alarm No to Alarm No Old
   #AlarmNo_Old := #AlarmNo;
END_REGION

REGION Network 133: Reset Ack Required
   IF (#AlarmNo = 0) OR #CMD_Acknowledge OR #FP_EN.Force THEN
       #ALARM_Failure_Ack_Requ := FALSE;
       #ALARM_Warn_Ack_Requ := FALSE;
   END_IF;
END_REGION

REGION Network 134: Skip = Skip Alarm
   IF (#AlarmNo = 0) OR #ALARM_Warn_Ack_Requ OR #ALARM_Failure_Ack_Requ THEN GOTO Skip; END_IF;
END_REGION

REGION Network 135: Clear Alarm
   Clr:
   #DummyBool := #DummyBool;
END_REGION

REGION Network 136: Clear Alarm
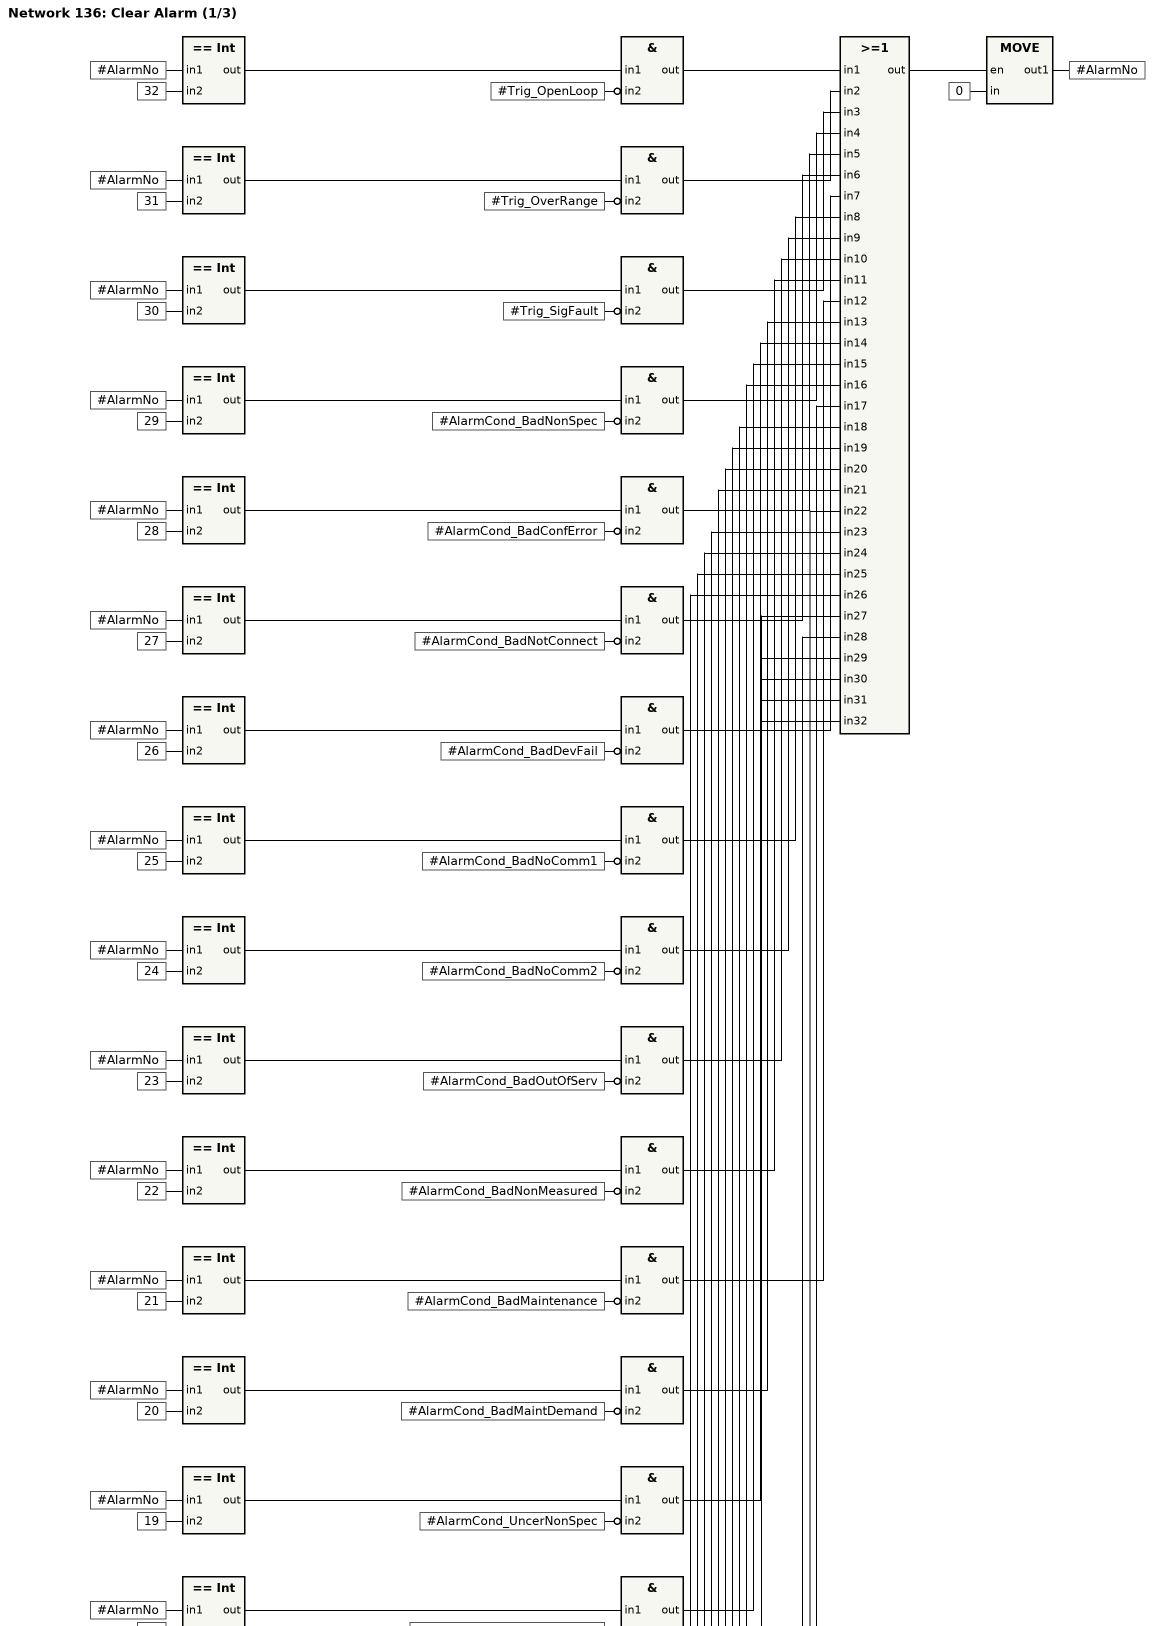
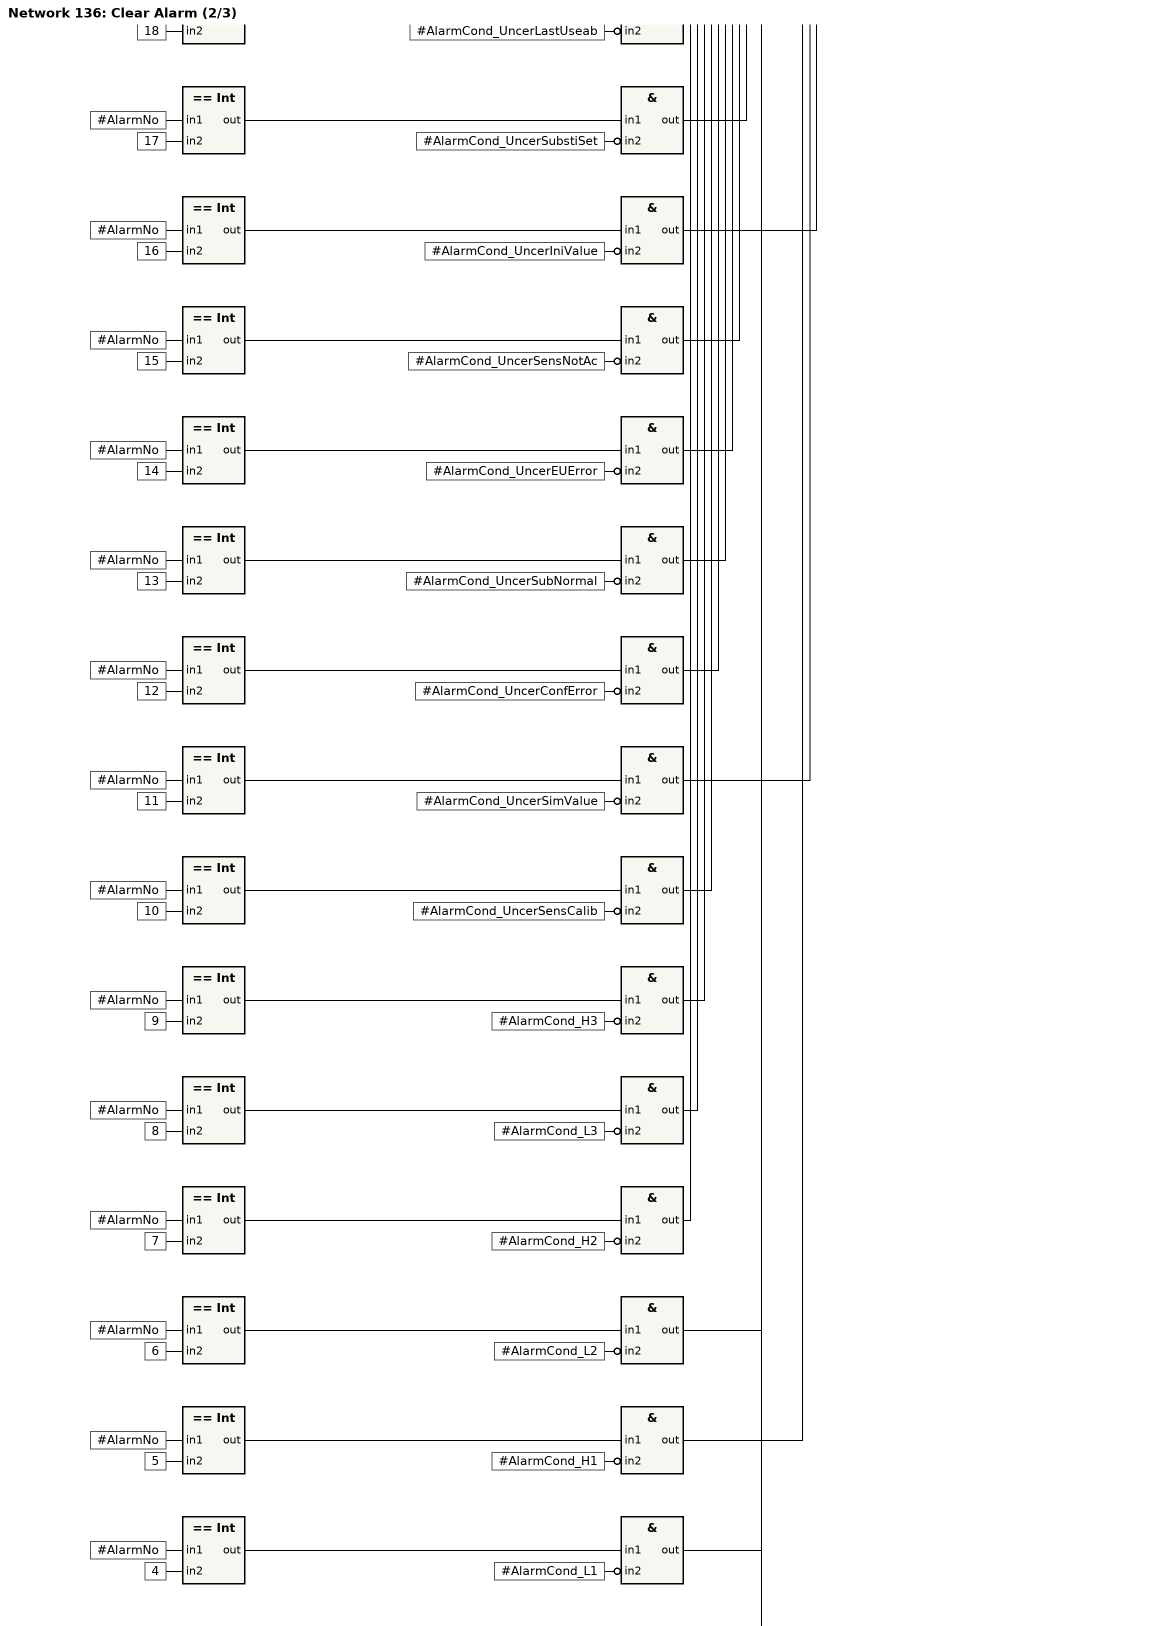
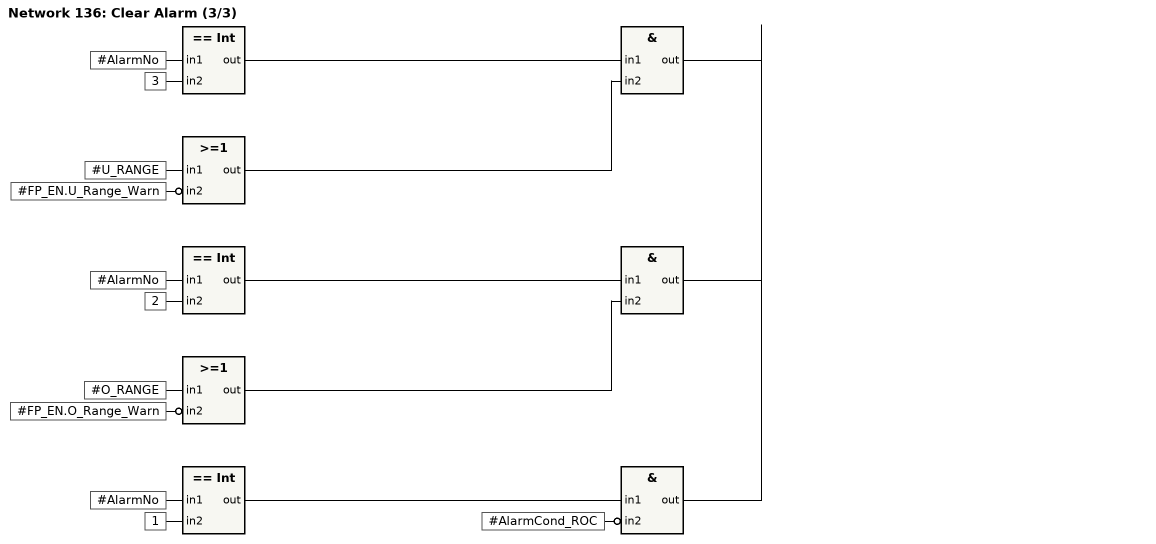
   IF ((#AlarmNo = 32) AND NOT #Trig_OpenLoop) OR ((#AlarmNo = 31) AND NOT #Trig_OverRange) OR ((#AlarmNo = 30) AND NOT #Trig_SigFault) OR ((#AlarmNo = 29) AND NOT #AlarmCond_BadNonSpec) OR ((#AlarmNo = 28) AND NOT #AlarmCond_BadConfError) OR ((#AlarmNo = 27) AND NOT #AlarmCond_BadNotConnect) OR ((#AlarmNo = 26) AND NOT #AlarmCond_BadDevFail) OR ((#AlarmNo = 25) AND NOT #AlarmCond_BadNoComm1) OR ((#AlarmNo = 24) AND NOT #AlarmCond_BadNoComm2) OR ((#AlarmNo = 23) AND NOT #AlarmCond_BadOutOfServ) OR ((#AlarmNo = 22) AND NOT #AlarmCond_BadNonMeasured) OR ((#AlarmNo = 21) AND NOT #AlarmCond_BadMaintenance) OR ((#AlarmNo = 20) AND NOT #AlarmCond_BadMaintDemand) OR ((#AlarmNo = 19) AND NOT #AlarmCond_UncerNonSpec) OR ((#AlarmNo = 18) AND NOT #AlarmCond_UncerLastUseab) OR ((#AlarmNo = 17) AND NOT #AlarmCond_UncerSubstiSet) OR ((#AlarmNo = 16) AND NOT #AlarmCond_UncerIniValue) OR ((#AlarmNo = 15) AND NOT #AlarmCond_UncerSensNotAc) OR ((#AlarmNo = 14) AND NOT #AlarmCond_UncerEUError) OR ((#AlarmNo = 13) AND NOT #AlarmCond_UncerSubNormal) OR ((#AlarmNo = 12) AND NOT #AlarmCond_UncerConfError) OR ((#AlarmNo = 11) AND NOT #AlarmCond_UncerSimValue) OR ((#AlarmNo = 10) AND NOT #AlarmCond_UncerSensCalib) OR ((#AlarmNo = 9) AND NOT #AlarmCond_H3) OR ((#AlarmNo = 8) AND NOT #AlarmCond_L3) OR ((#AlarmNo = 7) AND NOT #AlarmCond_H2) OR ((#AlarmNo = 6) AND NOT #AlarmCond_L2) OR ((#AlarmNo = 5) AND NOT #AlarmCond_H1) OR ((#AlarmNo = 4) AND NOT #AlarmCond_L1) OR ((#AlarmNo = 3) AND (#U_RANGE OR NOT #FP_EN.U_Range_Warn)) OR ((#AlarmNo = 2) AND (#O_RANGE OR NOT #FP_EN.O_Range_Warn)) OR ((#AlarmNo = 1) AND NOT #AlarmCond_ROC) THEN
       #AlarmNo := 0;
   END_IF;
END_REGION

REGION Network 137: Clear Alarm
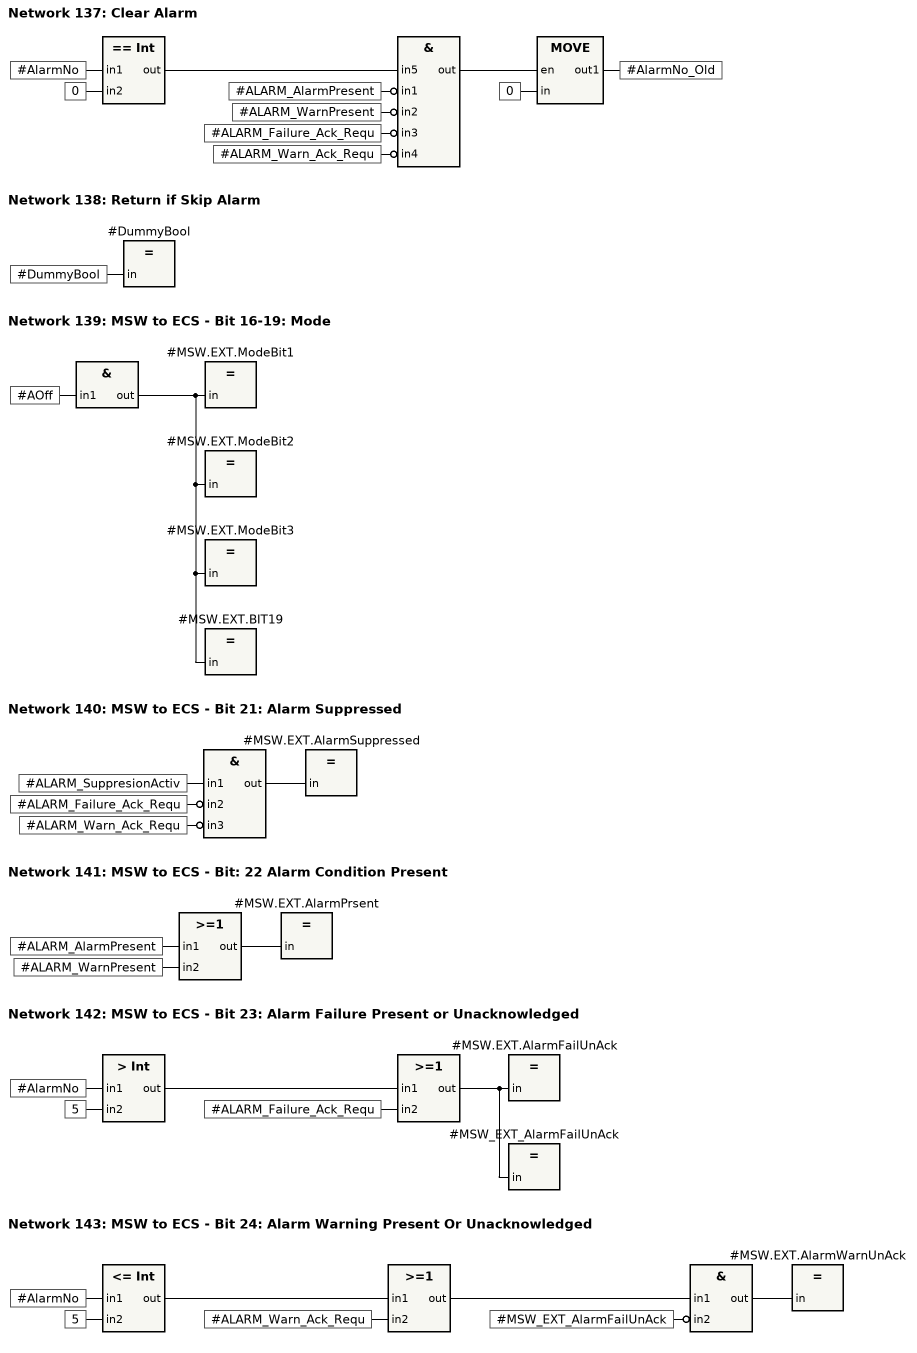
   IF (#AlarmNo = 0) AND NOT #ALARM_AlarmPresent AND NOT #ALARM_WarnPresent AND NOT #ALARM_Failure_Ack_Requ AND NOT #ALARM_Warn_Ack_Requ THEN
       #AlarmNo_Old := 0;
   END_IF;
END_REGION

REGION Network 138: Return if Skip Alarm
   Skip:
   #DummyBool := #DummyBool;
END_REGION

REGION Network 139: MSW to ECS - Bit 16-19: Mode
   // 0 = Auto
   // 1 = Single Start
   // 2 = Manual
   // 3 = Local
   // 4 = Test Mode
   #MSW.EXT.ModeBit1 := #AOff;
   #MSW.EXT.ModeBit2 := #AOff;
   #MSW.EXT.ModeBit3 := #AOff;
   #MSW.EXT.BIT19 := #AOff;
END_REGION

REGION Network 140: MSW to ECS - Bit 21: Alarm Suppressed
   #MSW.EXT.AlarmSuppressed := #ALARM_SuppresionActiv AND NOT #ALARM_Failure_Ack_Requ AND NOT #ALARM_Warn_Ack_Requ;
END_REGION

REGION Network 141: MSW to ECS - Bit: 22 Alarm Condition Present
   #MSW.EXT.AlarmPrsent := #ALARM_AlarmPresent OR #ALARM_WarnPresent;
END_REGION

REGION Network 142: MSW to ECS - Bit 23: Alarm Failure Present or Unacknowledged
   #MSW.EXT.AlarmFailUnAck := (#AlarmNo > 5) OR #ALARM_Failure_Ack_Requ;
   #MSW_EXT_AlarmFailUnAck := #MSW.EXT.AlarmFailUnAck;
END_REGION

REGION Network 143: MSW to ECS - Bit 24: Alarm Warning Present Or Unacknowledged
   #MSW.EXT.AlarmWarnUnAck := ((#AlarmNo <= 5) OR #ALARM_Warn_Ack_Requ) AND NOT #MSW_EXT_AlarmFailUnAck;
END_REGION

REGION Network 144: MSW to ECS - Bit 25: Acknowledge Required
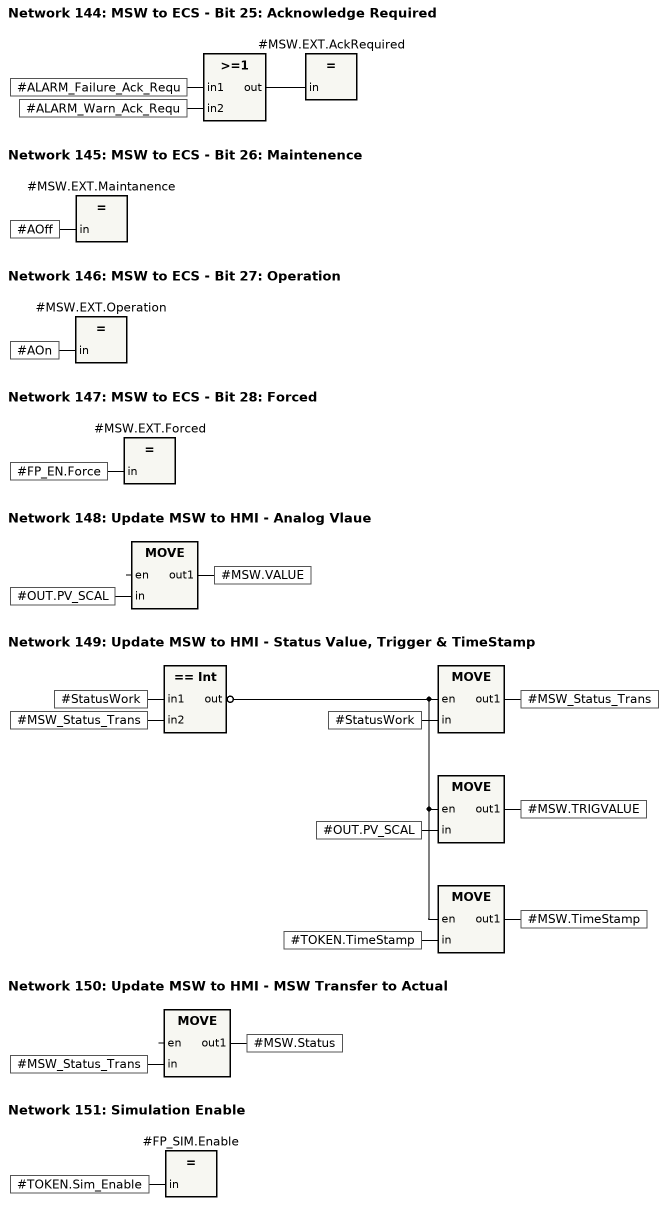
   #MSW.EXT.AckRequired := #ALARM_Failure_Ack_Requ OR #ALARM_Warn_Ack_Requ;
END_REGION

REGION Network 145: MSW to ECS - Bit 26: Maintenence
   #MSW.EXT.Maintanence := #AOff;
END_REGION

REGION Network 146: MSW to ECS - Bit 27: Operation
   // Build 004 - 22. Aug. 2016 (FKP) : #MSW.EXT.Operation set to constant on
   #MSW.EXT.Operation := #AOn;
END_REGION

REGION Network 147: MSW to ECS - Bit 28: Forced
   #MSW.EXT.Forced := #FP_EN.Force;
END_REGION

REGION Network 148: Update MSW to HMI - Analog Vlaue
   #MSW.VALUE := #OUT.PV_SCAL;
END_REGION

REGION Network 149: Update MSW to HMI - Status Value, Trigger & TimeStamp
   #_w1 := NOT (#StatusWork = #MSW_Status_Trans);
   IF #_w1 THEN
       #MSW_Status_Trans := #StatusWork;
       #MSW.TRIGVALUE := #OUT.PV_SCAL;
       #MSW.TimeStamp := #TOKEN.TimeStamp;
   END_IF;
END_REGION

REGION Network 150: Update MSW to HMI - MSW Transfer to Actual
   #MSW.Status := #MSW_Status_Trans;
END_REGION

REGION Network 151: Simulation Enable
   #FP_SIM.Enable := #TOKEN.Sim_Enable;
END_REGION

REGION Network 152: Simulation Enable
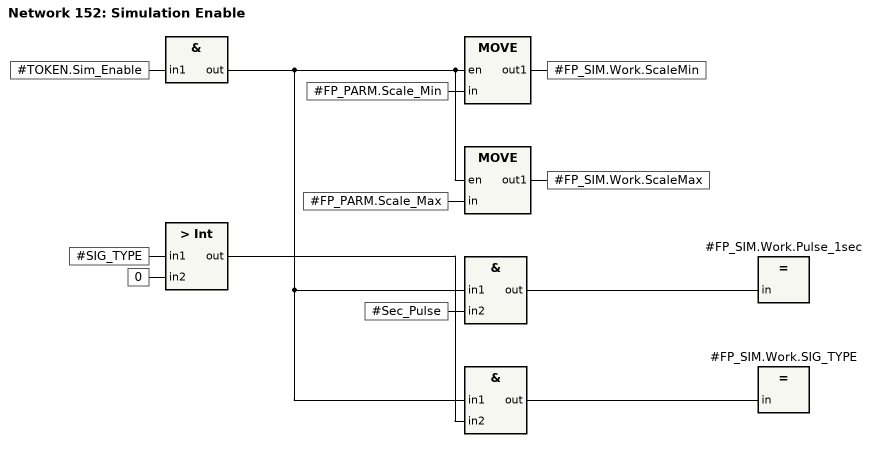
   IF #TOKEN.Sim_Enable THEN
       #FP_SIM.Work.ScaleMin := #FP_PARM.Scale_Min;
       #FP_SIM.Work.ScaleMax := #FP_PARM.Scale_Max;
   END_IF;
   #FP_SIM.Work.Pulse_1sec := #TOKEN.Sim_Enable AND #Sec_Pulse;
   #FP_SIM.Work.SIG_TYPE := #TOKEN.Sim_Enable AND (#SIG_TYPE > 0);
END_REGION

REGION Network 153: Write Stat to OUT
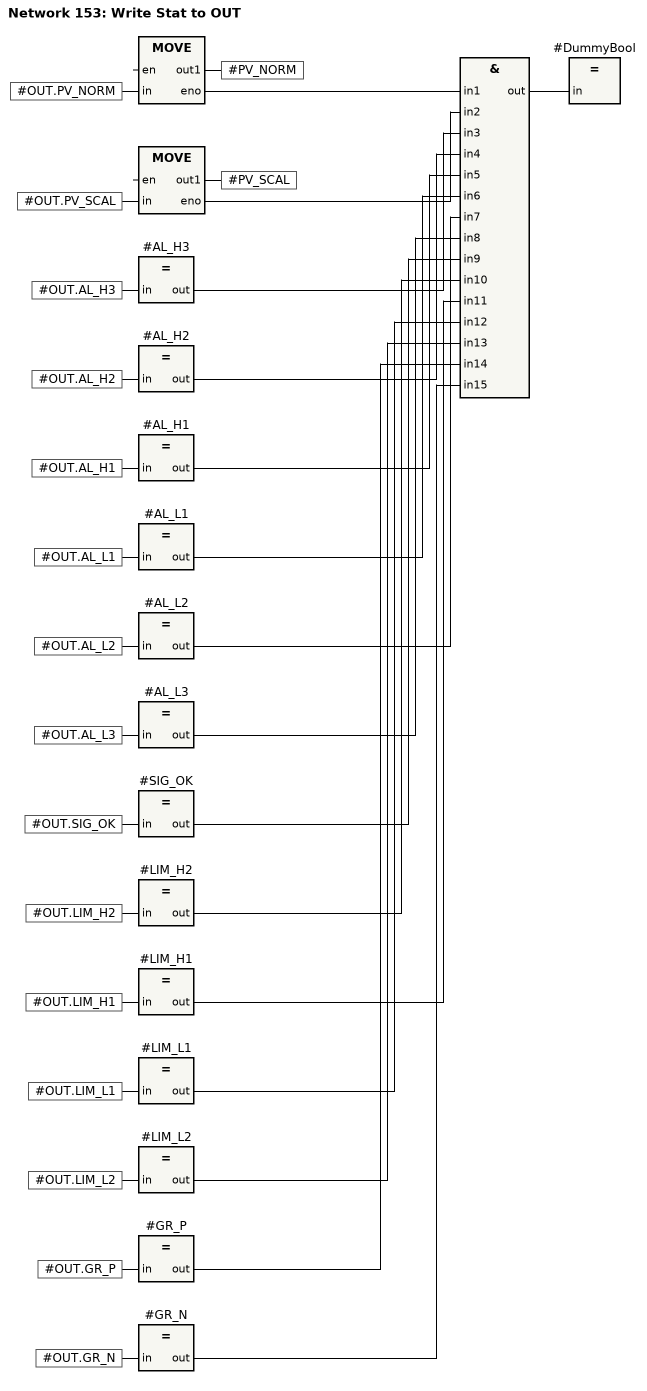
   #PV_NORM := #OUT.PV_NORM;
   #PV_SCAL := #OUT.PV_SCAL;
   #AL_H3 := #OUT.AL_H3;
   #AL_H2 := #OUT.AL_H2;
   #AL_H1 := #OUT.AL_H1;
   #AL_L1 := #OUT.AL_L1;
   #AL_L2 := #OUT.AL_L2;
   #AL_L3 := #OUT.AL_L3;
   #SIG_OK := #OUT.SIG_OK;
   #LIM_H2 := #OUT.LIM_H2;
   #LIM_H1 := #OUT.LIM_H1;
   #LIM_L1 := #OUT.LIM_L1;
   #LIM_L2 := #OUT.LIM_L2;
   #GR_P := #OUT.GR_P;
   #GR_N := #OUT.GR_N;
   #DummyBool := #OUT.AL_H3 AND #OUT.AL_H2 AND #OUT.AL_H1 AND #OUT.AL_L1 AND #OUT.AL_L2 AND #OUT.AL_L3 AND #OUT.SIG_OK AND #OUT.LIM_H2 AND #OUT.LIM_H1 AND #OUT.LIM_L1 AND #OUT.LIM_L2 AND #OUT.GR_P AND #OUT.GR_N;
END_REGION
END_FUNCTION_BLOCK

FUNCTION_BLOCK "ACESYS_SELECT"   // FB205, FBD
TITLE = ACESYS V8.0 - Build 001 - SELECT
{ S7_Optimized_Access := 'FALSE' }
AUTHOR : FLSmidth
FAMILY : ACESYS
NAME : SELECT
VERSION : 8.0
   VAR_INPUT
      ENAB : Bool := TRUE;   // Select Enable from Faceplate
      FCON : Bool;   // Select On
      FCOFF : Bool;   // Select off
   END_VAR
   VAR_OUTPUT
      SEL : Bool;   // Select on
      SELONS : Bool;   // Selct on oneshot
      SELOFFS : Bool;   // Select off oneshot
      MSW : "ACESYS_HMI_STAT_16";
   END_VAR
   VAR_IN_OUT
      TOKEN : "ACESYS_TOKEN";
   END_VAR
   VAR
      BlockInfo : Struct
         Ace_Version : Int;   // Acesys Block Version Number
         Ace_BuildNo : Int;   // Acesys Block Build Number
         State_Act : Int;   // Actual State Number
         State_Prev : Int;   // Previous State Number
         DB_Number : Int;   // Block Instance DB Number
      END_STRUCT;
      FP_CMD : Struct   // Faceplate Commands
         Spare_08 : Bool;
         Spare_09 : Bool;
         Spare_10 : Bool;
         Spare_11 : Bool;
         Spare_12 : Bool;
         Spare_13 : Bool;
         Spare_14 : Bool;
         AckAlarm : Bool;
         Toggle : Bool;   // Bit0
         Select : Bool;   // Bit1
         DeSelect : Bool;   // Bit2
         Inching : Bool;   // Bit3
         Spare_04 : Bool;
         Spare_05 : Bool;
         Spare_06 : Bool;
         Spare_07 : Bool;
      END_STRUCT;
      FP_DIM : Struct
         Select : Bool;
         Deselect : Bool;
      END_STRUCT;
      Ons_Sel : Bool;   // OneShoot Bit
      Ons_DeSel : Bool;   // OneShoot Bit
      Ons_FP_Sel : Bool;   // OneShoot Bit
      Ons_FP_DeSel : Bool;   // OneShoot Bit
      Ons_PosIncing : Bool;
      Ons_NegIncing : Bool;
      Spare10 : Bool;
      Spare09 : Bool;
      Spare08 : Bool;
      Spare07 : Bool;
      Spare06 : Bool;
      Spare05 : Bool;
      Spare04 : Bool;
      Spare03 : Bool;
      Spare02 : Bool;
      Spare01 : Bool;
      StatusWork : Int;
      OUT : Struct
         SEL : Bool;
         SELONS : Bool;
         SELOFFS : Bool;
      END_STRUCT;
      MSW_Status_Trans : Int;
   END_VAR
   VAR_TEMP
      Aon : Bool;
      Aoff : Bool;
      FP_Dim_Inching : Bool;
      DummyBool : Bool;
      ECSStatusBuilder : Int;
      MSW_Status : Int;
   END_VAR
   VAR_TEMP   // added for the SCL form of the ladder/FBD networks
      _w1 : Bool;
      _w2 : Bool;
      _w3 : Bool;
      _w4 : Bool;
   END_VAR
BEGIN

REGION Network 1: Always On
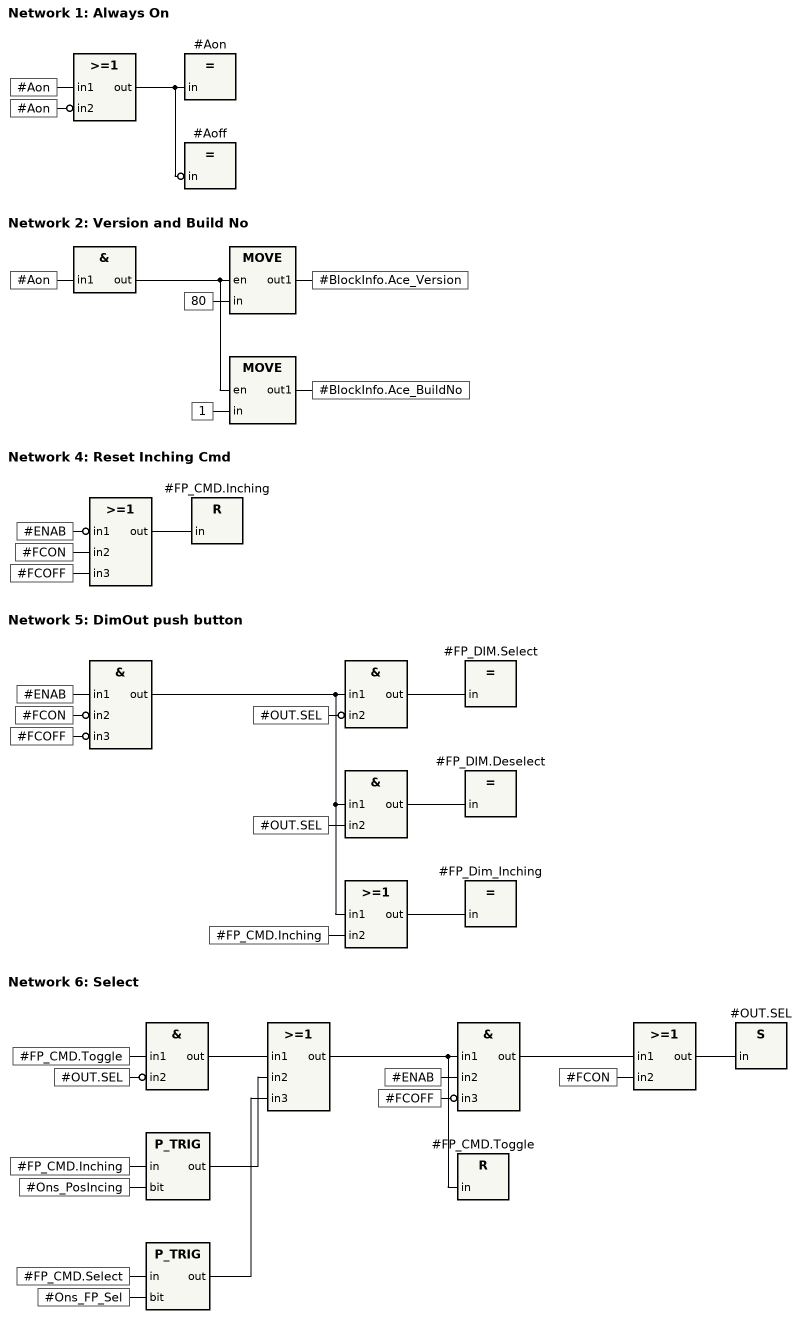
   #Aon := #Aon OR NOT #Aon;
   #Aoff := NOT #Aon;
END_REGION

REGION Network 2: Version and Build No
   IF #Aon THEN
       #BlockInfo.Ace_Version := 80;
       #BlockInfo.Ace_BuildNo := 1;
   END_IF;
END_REGION

REGION Network 3 (STL): Instance DB Number to Faceplate
         L     DINO;
         T     #BlockInfo.DB_Number;
END_REGION

REGION Network 4: Reset Inching Cmd
   IF NOT #ENAB OR #FCON OR #FCOFF THEN #FP_CMD.Inching := FALSE; END_IF;
END_REGION

REGION Network 5: DimOut push button
   #_w1 := #ENAB AND NOT #FCON AND NOT #FCOFF;
   #FP_DIM.Select := #_w1 AND NOT #OUT.SEL;
   #FP_DIM.Deselect := #_w1 AND #OUT.SEL;
   #FP_Dim_Inching := #_w1 OR #FP_CMD.Inching;
END_REGION

REGION Network 6: Select
   #_w1 := #FP_CMD.Inching AND NOT #Ons_PosIncing;   // rising edge
   #Ons_PosIncing := #FP_CMD.Inching;
   #_w2 := #FP_CMD.Select AND NOT #Ons_FP_Sel;   // rising edge
   #Ons_FP_Sel := #FP_CMD.Select;
   #_w3 := (#FP_CMD.Toggle AND NOT #OUT.SEL) OR #_w1 OR #_w2;
   IF (#_w3 AND #ENAB AND NOT #FCOFF) OR #FCON THEN #OUT.SEL := TRUE; END_IF;
   IF #_w3 THEN #FP_CMD.Toggle := FALSE; END_IF;
END_REGION

REGION Network 7: Deselect
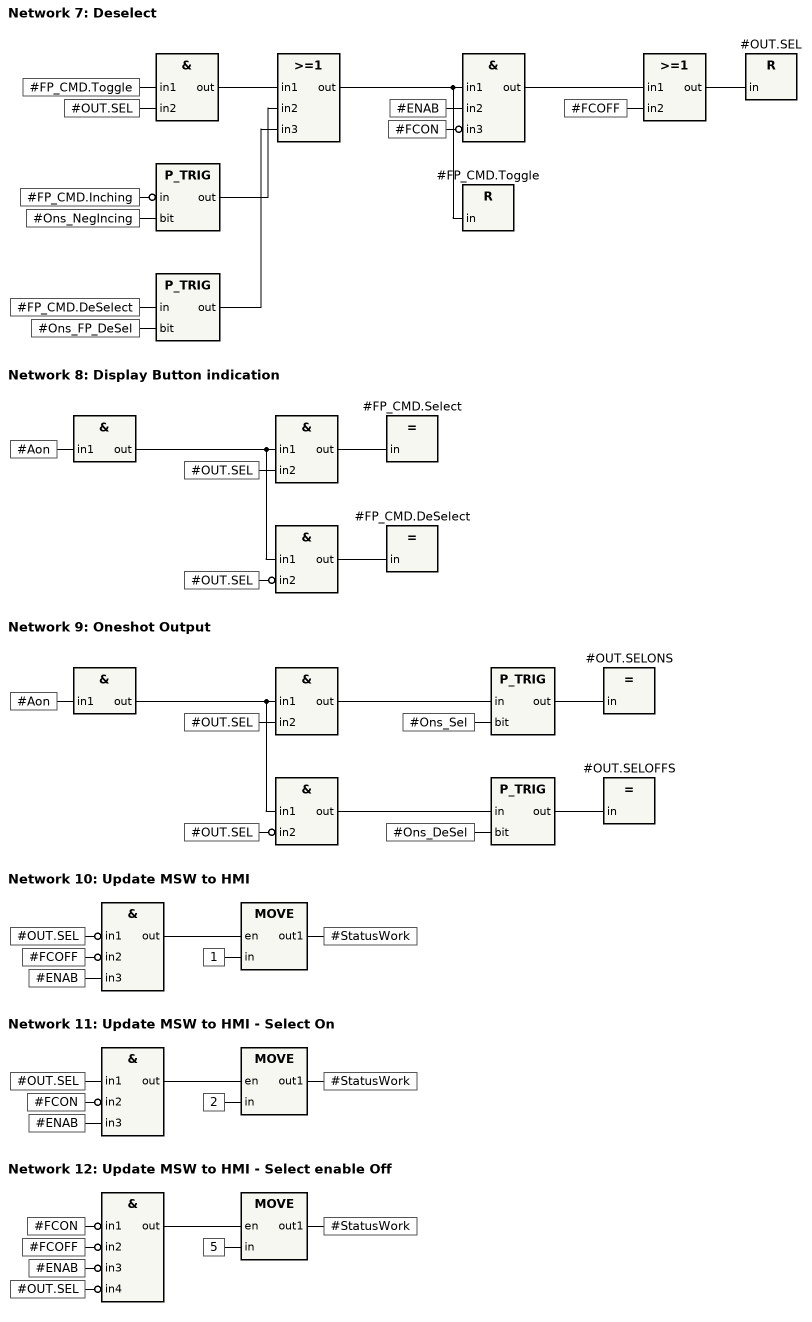
   #_w1 := NOT #FP_CMD.Inching AND NOT #Ons_NegIncing;   // rising edge
   #Ons_NegIncing := NOT #FP_CMD.Inching;
   #_w2 := #FP_CMD.DeSelect AND NOT #Ons_FP_DeSel;   // rising edge
   #Ons_FP_DeSel := #FP_CMD.DeSelect;
   #_w3 := (#FP_CMD.Toggle AND #OUT.SEL) OR #_w1 OR #_w2;
   IF (#_w3 AND #ENAB AND NOT #FCON) OR #FCOFF THEN #OUT.SEL := FALSE; END_IF;
   IF #_w3 THEN #FP_CMD.Toggle := FALSE; END_IF;
END_REGION

REGION Network 8: Display Button indication
   #FP_CMD.Select := #Aon AND #OUT.SEL;
   #FP_CMD.DeSelect := #Aon AND NOT #OUT.SEL;
END_REGION

REGION Network 9: Oneshot Output
   #_w1 := #Aon AND #OUT.SEL;
   #_w2 := #_w1 AND NOT #Ons_Sel;   // rising edge
   #Ons_Sel := #_w1;
   #OUT.SELONS := #_w2;
   #_w3 := #Aon AND NOT #OUT.SEL;
   #_w4 := #_w3 AND NOT #Ons_DeSel;   // rising edge
   #Ons_DeSel := #_w3;
   #OUT.SELOFFS := #_w4;
END_REGION

REGION Network 10: Update MSW to HMI
   IF NOT #OUT.SEL AND NOT #FCOFF AND #ENAB THEN #StatusWork := 1; END_IF;
END_REGION

REGION Network 11: Update MSW to HMI - Select On
   IF #OUT.SEL AND NOT #FCON AND #ENAB THEN #StatusWork := 2; END_IF;
END_REGION

REGION Network 12: Update MSW to HMI - Select enable Off
   IF NOT #FCON AND NOT #FCOFF AND NOT #ENAB AND NOT #OUT.SEL THEN #StatusWork := 5; END_IF;
END_REGION

REGION Network 13: Update MSW to HMI - Select enable On
